(*

short summary
=============

.. <legal notes>

legal notes
=================
| SPDX-FileCopyrightText: © 2023 ekvip automation GmbH <info@ekvip.de>
| SPDX-License-Identifier: Apache-2.0
| For details check: Apache-2.0_

.. _Apache-2.0: https://www.apache.org/licenses/LICENSE-2.0

.. </legal notes>

methods and properties
======================

*)

{warning 'header is generated please add your documentation'}
FUNCTION_BLOCK StringAssertionTests EXTENDS AbstractAssertorTest

VAR
	testDataStringLengthIsExact 	: ARRAY[0 ..IsLengthTestDataSet.SIZE_OF_IS_DATASET] OF IsLengthBasicData;
	testDataStringContains 			: ARRAY[0..containsTestDataSet.SIZE_OF_CONTAINS_DATASET] OF containsDataStr;
	testDataStringContainsNo 		: ARRAY[0..containsNOTestDataSet.SIZE_OF_CONTAINSNO_DATASET] OF containsDataStr;
	testDataStringStartsWith		: ARRAY[0..startsWithDataSet.SIZE_OF_STARTWITH_DATASET] OF containsDataStr;
	testDataStringEndsWith 			: ARRAY[0..endsWithDataSet.SIZE_OF_ENDSWITH_DATASET] OF containsDataStr;
	testDataStringIsEqual			: ARRAY[0..isEqualToTestDataSet.SIZE_OF_ISEQUALTO_DATASET] OF isEqualToDataStr;
	testDataStringIsNotEqual		: ARRAY[0..isNotEqualToTestDataSet.SIZE_OF_ISNOTEQUALTO_DATASET] OF isEqualToDataStr;
	testDataStringIsEmpty			: ARRAY[0..isEmptyTestDataSet.SIZE_OF_ISEMPTY_DATASET] OF isEmptyDataStr;
	testDataStringIsNotEmpty		: ARRAY[0..isNotEmtyTestDataSet.SIZE_OF_ISNOTEMPTY_DATASET] OF isEmptyDataStr;
	testDataStringIsLenghtBetween	: ARRAY[0..IsLengthBetweenDataSet.SIZE_OF_LENGTHBETWEEN_DATASET] OF IsLengthBetweenBasicData;
	
END_VAR

testAnyString_isEmpty();
testAnyString_isNotEmpty();
testAnyString_isEqualTo();
testAnyString_isNotEqualTo();
testAnyString_lengthIsExact();


THIS^.runTestIsLength();
THIS^.runTestContains();
THIS^.runTestContainsNo();
THIS^.runTestEndsWith();
THIS^.runTestStartsWith();
THIS^.runTestIsEmpty();
THIS^.runTestIsNotEmpty();
THIS^.runTestIsEqualTo();
THIS^.runTestIsNotEqualTo();
THIS^.runTestLengthIsBetween();

(*

short summary
=============

.. <legal notes>

legal notes
=================
| SPDX-FileCopyrightText: © 2023 ekvip automation GmbH <info@ekvip.de>
| SPDX-License-Identifier: Apache-2.0
| For details check: Apache-2.0_

.. _Apache-2.0: https://www.apache.org/licenses/LICENSE-2.0

.. </legal notes>

parameters
==========

*)

{warning 'header is generated please add your documentation'}
METHOD FB_init : BOOL
VAR_INPUT
    bInitRetains : BOOL; // if TRUE, the retain variables are initialized (warm start / cold start)
    bInCopyCode : BOOL;  // if TRUE, the instance afterwards gets moved into the copy code (online change)
	classToBeTested :IAssertorContainer;
END_VAR
THIS^.testDataStringLengthIsExact 	:= IsLengthTestDataSet.IsLenghtDataSetCommon;
THIS^.testDataStringContains 		:= containsTestDataSet.containsDataSetCommon;	
THIS^.testDataStringContainsNo		:= containsNoTestDataSet.containsNoDataSetCommon;
THIS^.testDataStringEndsWith		:= endsWithDataSet.endsWithDataSetCommon;
THIS^.testDataStringStartsWith		:= startsWithDataSet.StartsWithDataSetCommon;
THIS^.testDataStringIsEqual			:= isEqualToTestDataSet.isEqualToDataSetCommon;		
THIS^.testDataStringIsNotEqual		:= isNotEqualToTestDataSet.isNotEqualDataSetCommon;
THIS^.testDataStringIsEmpty			:= isEmptyTestDataSet.isEmptyDataSetCommon;
THIS^.testDataStringIsNotEmpty		:= isNotEmtyTestDataSet.isNotEmptyDataSetCommon;
THIS^.testDataStringIsLenghtBetween	:= IsLengthBetweenDataSet.isLenghtBetweenToDataSetCommon;
END_METHOD

(*

short summary
=============

.. <legal notes>

legal notes
=================
| SPDX-FileCopyrightText: © 2023 ekvip automation GmbH <info@ekvip.de>
| SPDX-License-Identifier: Apache-2.0
| For details check: Apache-2.0_

.. _Apache-2.0: https://www.apache.org/licenses/LICENSE-2.0

.. </legal notes>

parameters
==========

*)

{warning 'header is generated please add your documentation'}
METHOD reset
VAR_INPUT
END_VAR
THIS^.assertorContainer.resetAssertor();
END_METHOD

(*

short summary
=============

.. <legal notes>

legal notes
=================
| SPDX-FileCopyrightText: © 2023 ekvip automation GmbH <info@ekvip.de>
| SPDX-License-Identifier: Apache-2.0
| For details check: Apache-2.0_

.. _Apache-2.0: https://www.apache.org/licenses/LICENSE-2.0

.. </legal notes>

parameters
==========

*)

{warning 'header is generated please add your documentation'}
METHOD runTestContains
VAR
	testDataIterator	:USINT;
END_VAR
TEST('ContainsTests');
FOR testDataIterator := 0 TO containsTestDataSet.SIZE_OF_contains_DATASET DO
	IF (THIS^.testDataStringContains[testDataIterator].typeToTest = TypeToTest.TEST_STRING) THEN
		
		THIS^.testAnyStringContains(THIS^.testDataStringContains[testDataIterator], testDataIterator);
		THIS^.testAsciiStringContains (THIS^.testDataStringContains[testDataIterator], testDataIterator);
		
	ELSIF (THIS^.testDataStringContains[testDataIterator].typeToTest = TypeToTest.TEST_WSTRING) THEN
		
		THIS^.testAnyStringContains(THIS^.testDataStringContains[testDataIterator], testDataIterator);
		THIS^.testUtf16StringContains(THIS^.testDataStringContains[testDataIterator], testDataIterator);
		
	END_IF;
END_FOR

TEST_FINISHED();
END_METHOD

(*

short summary
=============

.. <legal notes>

legal notes
=================
| SPDX-FileCopyrightText: © 2023 ekvip automation GmbH <info@ekvip.de>
| SPDX-License-Identifier: Apache-2.0
| For details check: Apache-2.0_

.. _Apache-2.0: https://www.apache.org/licenses/LICENSE-2.0

.. </legal notes>

parameters
==========

*)

{warning 'header is generated please add your documentation'}
METHOD runTestContainsNo
VAR
	testDataIterator	:USINT;
END_VAR
TEST('ContainsNoTests');
FOR testDataIterator:= 0 TO containsNoTestDataSet.SIZE_OF_containsNo_DATASET DO
	IF (THIS^.testDataStringContainsNo[testDataIterator].typeToTest = TypeToTest.TEST_STRING) THEN
		
		THIS^.testAnyStringContainsNo(THIS^.testDataStringContainsno[testDataIterator], testDataIterator);
		THIS^.testAsciiStringContainsNo (THIS^.testDataStringContainsno[testDataIterator], testDataIterator);
		
	ELSIF (THIS^.testDataStringContainsNo[testDataIterator].typeToTest = TypeToTest.TEST_WSTRING) THEN
		
		THIS^.testAnyStringContainsNo(THIS^.testDataStringContainsno[testDataIterator], testDataIterator);
		THIS^.testUtf16StringContainsNo(THIS^.testDataStringContainsno[testDataIterator], testDataIterator);
		
	END_IF;
END_FOR

TEST_FINISHED();
END_METHOD

(*

short summary
=============

.. <legal notes>

legal notes
=================
| SPDX-FileCopyrightText: © 2023 ekvip automation GmbH <info@ekvip.de>
| SPDX-License-Identifier: Apache-2.0
| For details check: Apache-2.0_

.. _Apache-2.0: https://www.apache.org/licenses/LICENSE-2.0

.. </legal notes>

parameters
==========

*)

{warning 'header is generated please add your documentation'}
METHOD runTestEndsWith
VAR
	testDataIterator	: USINT;
END_VAR
TEST('endsWithTests');

FOR testDataIterator := 0 TO endsWithDataSet.SIZE_OF_ENDSWITH_DATASET DO
	IF (THIS^.testDataStringEndsWith[testDataIterator].typeToTest = TypeToTest.TEST_STRING) THEN
		
		THIS^.testAnyStringEndsWith(THIS^.testDataStringEndsWith[testDataIterator], testDataIterator);
		THIS^.testAsciiEndsWith(THIS^.testDataStringEndsWith[testDataIterator], testDataIterator);
		
	ELSIF (THIS^.testDataStringEndsWith[testDataIterator].typeToTest = TypeToTest.TEST_WSTRING) THEN
		
		THIS^.testAnyStringEndsWith(THIS^.testDataStringEndsWith[testDataIterator], testDataIterator);
		THIS^.testUtf16EndsWith(THIS^.testDataStringEndsWith[testDataIterator], testDataIterator);
		
	END_IF;
END_FOR

TEST_FINISHED();
END_METHOD

(*

short summary
=============

.. <legal notes>

legal notes
=================
| SPDX-FileCopyrightText: © 2023 ekvip automation GmbH <info@ekvip.de>
| SPDX-License-Identifier: Apache-2.0
| For details check: Apache-2.0_

.. _Apache-2.0: https://www.apache.org/licenses/LICENSE-2.0

.. </legal notes>

parameters
==========

*)

{warning 'header is generated please add your documentation'}
METHOD runTestIsEmpty
VAR
	testDataIterator	: USINT;
END_VAR
TEST('isEmptyTests');

FOR testDataIterator := 0 TO isEmptyTestDataSet.SIZE_OF_ISEMPTY_DATASET DO
	IF (THIS^.testDataStringIsEmpty[testDataIterator].typeToTest = TypeToTest.TEST_STRING) THEN
		
		THIS^.testAnyStringIsEmpty(THIS^.testDataStringIsEmpty[testDataIterator], testDataIterator);
		THIS^.testAsciiIsEmpty(THIS^.testDataStringIsEmpty[testDataIterator], testDataIterator);
		
	ELSIF (THIS^.testDataStringIsEmpty[testDataIterator].typeToTest = TypeToTest.TEST_WSTRING) THEN
		
		THIS^.testAnyStringIsEmpty(THIS^.testDataStringIsEmpty[testDataIterator], testDataIterator);
		THIS^.testUtf16IsEmpty(THIS^.testDataStringIsEmpty[testDataIterator], testDataIterator);
		
	END_IF;
END_FOR

TEST_FINISHED();
END_METHOD

(*

short summary
=============

.. <legal notes>

legal notes
=================
| SPDX-FileCopyrightText: © 2023 ekvip automation GmbH <info@ekvip.de>
| SPDX-License-Identifier: Apache-2.0
| For details check: Apache-2.0_

.. _Apache-2.0: https://www.apache.org/licenses/LICENSE-2.0

.. </legal notes>

parameters
==========

*)

{warning 'header is generated please add your documentation'}
METHOD runTestIsEqualTo
VAR
	testDataIterator	: USINT;
END_VAR
TEST('isEqualToTests');

FOR testDataIterator := 0 TO isEqualToTestDataSet.SIZE_OF_ISEQUALTO_DATASET DO
	IF (THIS^.testDataStringIsEqual[testDataIterator].typeToTest = TypeToTest.TEST_STRING) THEN
		
		THIS^.testAnyStringIsEqualTo(THIS^.testDataStringIsEqual[testDataIterator], testDataIterator);
		THIS^.testAsciiIsEqualTo(THIS^.testDataStringIsEqual[testDataIterator], testDataIterator);
		
	ELSIF (THIS^.testDataStringIsEqual[testDataIterator].typeToTest = TypeToTest.TEST_WSTRING) THEN
		
		THIS^.testAnyStringIsEqualTo(THIS^.testDataStringIsEqual[testDataIterator], testDataIterator);
		THIS^.testUtf16IsEqualTo(THIS^.testDataStringIsEqual[testDataIterator], testDataIterator);
		
	END_IF;
END_FOR

TEST_FINISHED();
END_METHOD

(*

short summary
=============

.. <legal notes>

legal notes
=================
| SPDX-FileCopyrightText: © 2023 ekvip automation GmbH <info@ekvip.de>
| SPDX-License-Identifier: Apache-2.0
| For details check: Apache-2.0_

.. _Apache-2.0: https://www.apache.org/licenses/LICENSE-2.0

.. </legal notes>

parameters
==========

*)

{warning 'header is generated please add your documentation'}
METHOD runTestIsLength
VAR
	testDataIterator	:USINT;
END_VAR
TEST('IsLenghtIsTests');
FOR testDataIterator:= 0 TO IsLengthTestDataSet.SIZE_OF_IS_DATASET DO
	IF (THIS^.testDataStringLengthIsExact[testDataIterator].typeToTest = TypeToTest.TEST_STRING) THEN
		
		THIS^.testAnyStringLengthIs(THIS^.testDataStringLengthIsExact[testDataIterator], testDataIterator);
		THIS^.testAsciiStringlengthIs (THIS^.testDataStringLengthIsExact[testDataIterator], testDataIterator);
		
	ELSIF (THIS^.testDataStringLengthIsExact[testDataIterator].typeToTest = TypeToTest.TEST_WSTRING) THEN
		
		THIS^.testAnyStringLengthIs(THIS^.testDataStringLengthIsExact[testDataIterator], testDataIterator);
		THIS^.testUtf16StringlengthIs(THIS^.testDataStringLengthIsExact[testDataIterator], testDataIterator);
		
	END_IF;
END_FOR

TEST_FINISHED();
END_METHOD

(*

short summary
=============

.. <legal notes>

legal notes
=================
| SPDX-FileCopyrightText: © 2023 ekvip automation GmbH <info@ekvip.de>
| SPDX-License-Identifier: Apache-2.0
| For details check: Apache-2.0_

.. _Apache-2.0: https://www.apache.org/licenses/LICENSE-2.0

.. </legal notes>

parameters
==========

*)

{warning 'header is generated please add your documentation'}
METHOD runTestIsNotEmpty
VAR
	testDataIterator	: USINT;
END_VAR
TEST('isNotEmptyTests');

FOR testDataIterator := 0 TO isNotEmtyTestDataSet.SIZE_OF_ISNOTEMPTY_DATASET DO
	IF (THIS^.testDataStringIsNotEmpty[testDataIterator].typeToTest = TypeToTest.TEST_STRING) THEN
		
		THIS^.testAnyStringIsNotEmpty(THIS^.testDataStringIsNotEmpty[testDataIterator], testDataIterator);
		THIS^.testAsciiIsNotEmpty(THIS^.testDataStringIsNotEmpty[testDataIterator], testDataIterator);
		
	ELSIF (THIS^.testDataStringIsNotEmpty[testDataIterator].typeToTest = TypeToTest.TEST_WSTRING) THEN
		
		THIS^.testAnyStringIsNotEmpty(THIS^.testDataStringIsNotEmpty[testDataIterator], testDataIterator);
		THIS^.testUtf16IsNotEmpty(THIS^.testDataStringIsNotEmpty[testDataIterator], testDataIterator);
		
	END_IF;
END_FOR

TEST_FINISHED();
END_METHOD

(*

short summary
=============

.. <legal notes>

legal notes
=================
| SPDX-FileCopyrightText: © 2023 ekvip automation GmbH <info@ekvip.de>
| SPDX-License-Identifier: Apache-2.0
| For details check: Apache-2.0_

.. _Apache-2.0: https://www.apache.org/licenses/LICENSE-2.0

.. </legal notes>

parameters
==========

*)

{warning 'header is generated please add your documentation'}
METHOD runTestIsNotEqualTo
VAR
	testDataIterator	: USINT;
END_VAR
TEST('isNotEqualToTests');

FOR testDataIterator := 0 TO isNotEqualToTestDataSet.SIZE_OF_ISNOTEQUALTO_DATASET DO
	IF (THIS^.testDataStringIsNotEqual[testDataIterator].typeToTest = TypeToTest.TEST_STRING) THEN
		
		THIS^.testAnyStringIsNotEqualTo(THIS^.testDataStringIsNotEqual[testDataIterator], testDataIterator);
		THIS^.testAsciiIsNotEqualTo(THIS^.testDataStringIsNotEqual[testDataIterator], testDataIterator);
		
	ELSIF (THIS^.testDataStringIsNotEqual[testDataIterator].typeToTest = TypeToTest.TEST_WSTRING) THEN
		
		THIS^.testAnyStringIsNotEqualTo(THIS^.testDataStringIsNotEqual[testDataIterator], testDataIterator);
		THIS^.testUtf16IsNotEqualTo(THIS^.testDataStringIsNotEqual[testDataIterator], testDataIterator);
		
	END_IF;
END_FOR

TEST_FINISHED();
END_METHOD

(*

short summary
=============

.. <legal notes>

legal notes
=================
| SPDX-FileCopyrightText: © 2023 ekvip automation GmbH <info@ekvip.de>
| SPDX-License-Identifier: Apache-2.0
| For details check: Apache-2.0_

.. _Apache-2.0: https://www.apache.org/licenses/LICENSE-2.0

.. </legal notes>

parameters
==========

*)

{warning 'header is generated please add your documentation'}
METHOD runTestLengthIsBetween : BOOL
VAR
	testDataIterator	:USINT;
END_VAR
TEST('IsLenghtBetweenTests');
FOR testDataIterator:= 0 TO IsLengthBetweenDataSet.SIZE_OF_LENGTHBETWEEN_DATASET DO
	IF (THIS^.testDataStringIsLenghtBetween[testDataIterator].typeToTest = TypeToTest.TEST_STRING) THEN
		
		THIS^.testAnyStringLengthBetween(THIS^.testDataStringIsLenghtBetween[testDataIterator], testDataIterator);
		THIS^.testAsciiStringLengthBetween (THIS^.testDataStringIsLenghtBetween[testDataIterator], testDataIterator);
		
	ELSIF (THIS^.testDataStringIsLenghtBetween[testDataIterator].typeToTest = TypeToTest.TEST_WSTRING) THEN
		
		THIS^.testAnyStringLengthBetween(THIS^.testDataStringIsLenghtBetween[testDataIterator], testDataIterator);
		THIS^.testUtf16StringLengthBetween(THIS^.testDataStringIsLenghtBetween[testDataIterator], testDataIterator);
		
	END_IF;
END_FOR

TEST_FINISHED();
END_METHOD

(*

short summary
=============

.. <legal notes>

legal notes
=================
| SPDX-FileCopyrightText: © 2023 ekvip automation GmbH <info@ekvip.de>
| SPDX-License-Identifier: Apache-2.0
| For details check: Apache-2.0_

.. _Apache-2.0: https://www.apache.org/licenses/LICENSE-2.0

.. </legal notes>

parameters
==========

*)

{warning 'header is generated please add your documentation'}
METHOD runTestStartsWith
VAR
	testDataIterator	: USINT;
END_VAR
TEST('StartsWithTests');
FOR testDataIterator := 0 TO startsWithDataSet.SIZE_OF_STARTWITH_DATASET DO
	IF (THIS^.testDataStringStartsWith[testDataIterator].typeToTest = TypeToTest.TEST_STRING) THEN
		
		THIS^.testAnyStringStartsWith(THIS^.testDataStringStartsWith[testDataIterator], testDataIterator);
		THIS^.testAsciiStartsWith(THIS^.testDataStringStartsWith[testDataIterator], testDataIterator);
		
	ELSIF (THIS^.testDataStringStartsWith[testDataIterator].typeToTest = TypeToTest.TEST_WSTRING) THEN
		
		THIS^.testAnyStringStartsWith(THIS^.testDataStringStartsWith[testDataIterator], testDataIterator);
		THIS^.testUtf16StartsWith(THIS^.testDataStringStartsWith[testDataIterator], testDataIterator);
		
	END_IF;
END_FOR

TEST_FINISHED();
END_METHOD

(*

short summary
=============

.. <legal notes>

legal notes
=================
| SPDX-FileCopyrightText: © 2023 ekvip automation GmbH <info@ekvip.de>
| SPDX-License-Identifier: Apache-2.0
| For details check: Apache-2.0_

.. _Apache-2.0: https://www.apache.org/licenses/LICENSE-2.0

.. </legal notes>

parameters
==========

*)

{warning 'header is generated please add your documentation'}
METHOD testAnyString_isEmpty

VAR 
  testString1: STRING(50);
  testString2: STRING;
  number: INT;
END_VAR

// anyStringAssertionTests.isEmpty Tests

//-------------------------------------------------------------------------------------------------------
TEST('anyStringAssertionTest.isEmpty with stringToCheck:= emptyString');

testString1:= '';
THIS^.assertorContainer.resetAssertor();
THIS^.assertorContainer.assertor.assert.strings.anyString.isEmpty(
  stringToCheck := testString1,
  message := ''
);
THIS^.AssertFalse(
	Condition := THIS^.assertorContainer.wasAssertionWrong,
	Message := 'anyStringAssertionTests.isEmpty assertion shall be wrong, stringToCheck:= emptyString '
);
TEST_FINISHED();

//-------------------------------------------------------------------------------------------------------

TEST('anyStringAssertionTest.isEmpty with stringToCheck:= space');

testString1:= ' ';
THIS^.assertorContainer.resetAssertor();
THIS^.assertorContainer.assertor.assert.strings.anyString.isEmpty(
  stringToCheck := testString1,
  message := ''
);
THIS^.AssertTrue(
	Condition := THIS^.assertorContainer.wasAssertionWrong,
	Message := 'anyStringAssertionTests.isEmpty assertion shall be wrong, stringToCheck:= just space'
);
TEST_FINISHED();

//-------------------------------------------------------------------------------------------------------

TEST('anyStringAssertionTest.isEmpty with stringToCheck:= point');

testString1:= '.';
THIS^.assertorContainer.resetAssertor();
THIS^.assertorContainer.assertor.assert.strings.anyString.isEmpty(
  stringToCheck := testString1,
  message := ''
);
THIS^.AssertTrue(
	Condition := THIS^.assertorContainer.wasAssertionWrong,
	Message := 'anyStringAssertionTests.isEmpty assertion shall be wrong, stringToCheck:= point'
);
TEST_FINISHED();

//-------------------------------------------------------------------------------------------------------

TEST('anyStringAssertionTest.isEmpty with stringToCheck:= emptyStringVar');

testString1:= testString2;
THIS^.assertorContainer.resetAssertor();
THIS^.assertorContainer.assertor.assert.strings.anyString.isEmpty(
  stringToCheck := testString1,
  message := ''
);
THIS^.AssertFalse(
	Condition := THIS^.assertorContainer.wasAssertionWrong,
	Message := 'anyStringAssertionTests.isEmpty assertion shall be wrong, stringToCheck:= emptyStringVar'
);
TEST_FINISHED();

//-------------------------------------------------------------------------------------------------------

TEST('anyStringAssertionTest.isEmpty with stringToCheck:= wierdString');

testString1:= 'sadhasdhasduhuiashdui';
THIS^.assertorContainer.resetAssertor();
THIS^.assertorContainer.assertor.assert.strings.anyString.isEmpty(
  stringToCheck := testString1,
  message := ''
);
THIS^.AssertTrue(
	Condition := THIS^.assertorContainer.wasAssertionWrong,
	Message := 'anyStringAssertionTests.isEmpty assertion shall be wrong, stringToCheck:= emptyStringVar'
);
TEST_FINISHED();

//-------------------------------------------------------------------------------------------------------

TEST('anyStringAssertionTest.isEmpty with stringToCheck:=   +gdjsnd.8959889mfknfji');

testString1:= '   +gdjsnd.8959889mfknfji';
THIS^.assertorContainer.resetAssertor();
THIS^.assertorContainer.assertor.assert.strings.anyString.isEmpty(
  stringToCheck := testString1,
  message := ''
);
THIS^.AssertTrue(
	Condition := THIS^.assertorContainer.wasAssertionWrong,
	Message := 'anyStringAssertionTests.isEmpty assertion shall be wrong, stringToCheck:= emptyStringVar'
);
TEST_FINISHED();

//-------------------------------------------------------------------------------------------------------

TEST('anyStringAssertionTest.isEmpty with stringToCheck:=   converted int');

testString1:= INT_TO_STRING(number);
THIS^.assertorContainer.resetAssertor();
THIS^.assertorContainer.assertor.assert.strings.anyString.isEmpty(
  stringToCheck := testString1,
  message := ''
);
THIS^.AssertTrue(
	Condition := THIS^.assertorContainer.wasAssertionWrong,
	Message := 'anyStringAssertionTests.isEmpty assertion shall be wrong, stringToCheck:=  converted int'
);
TEST_FINISHED();
END_METHOD

(*

short summary
=============

.. <legal notes>

legal notes
=================
| SPDX-FileCopyrightText: © 2023 ekvip automation GmbH <info@ekvip.de>
| SPDX-License-Identifier: Apache-2.0
| For details check: Apache-2.0_

.. _Apache-2.0: https://www.apache.org/licenses/LICENSE-2.0

.. </legal notes>

parameters
==========

*)

{warning 'header is generated please add your documentation'}
METHOD testAnyString_isEqualTo

VAR 
  testString1: STRING(50);
  testString2: STRING(30);
  testString3: WSTRING(50);
  testString4: STRING(50);
  testString5: WSTRING(400);
  testString6: WSTRING(400);
  number: INT;
END_VAR

// anyStringAssertionTests.isEqualTo Tests

//-------------------------------------------------------------------------------------------------------
TEST('anyStringAssertionTest.isEqualTo with stringToCheck:= emptyString , expected:= emptyString , ignoreCases:= TRUE ,');

THIS^.assertorContainer.resetAssertor();
THIS^.assertorContainer.assertor.assert.strings.anyString.isEqualTo(
  stringToCheck:= testString1 , 
  expected:= testString2 ,
  ignoreCases:= TRUE ,
  message:='' );
  
THIS^.AssertFalse(
	Condition := THIS^.assertorContainer.wasAssertionWrong,
	Message := 'anyStringAssertionTests.isEqualTo , stringToCheck:= emptyString , expected:= emptyString , ignoreCases:= TRUE '
);
TEST_FINISHED();

//-------------------------------------------------------------------------------------------------------
TEST('anyStringAssertionTest.isEqualTo with stringToCheck:= emptyString assign , expected:= emptyString assign , ignoreCases:= TRUE ,');

testString1:= '';
testString2:= '';

THIS^.assertorContainer.resetAssertor();
THIS^.assertorContainer.assertor.assert.strings.anyString.isEqualTo(
  stringToCheck:= testString1 , 
  expected:= testString2 ,
  ignoreCases:= TRUE ,
  message:='' );
  
THIS^.AssertFalse(
	Condition := THIS^.assertorContainer.wasAssertionWrong,
	Message := 'anyStringAssertionTests.isEqualTo , stringToCheck:= emptyString assign, expected:= emptyString assign , ignoreCases:= TRUE '
);
TEST_FINISHED();

//-------------------------------------------------------------------------------------------------------
TEST('anyStringAssertionTest.isEqualTo with stringToCheck:= abcd56ä² , expected:= abcd56ä2 , ignoreCases:= TRUE ,');

testString1:= 'abcd56ä²';
testString2:= 'abcd56ä2';

THIS^.assertorContainer.resetAssertor();
THIS^.assertorContainer.assertor.assert.strings.anyString.isEqualTo(
  stringToCheck:= testString1 , 
  expected:= testString2 ,
  ignoreCases:= TRUE ,
  message:='' );
  
THIS^.AssertTrue(
	Condition := THIS^.assertorContainer.wasAssertionWrong,
	Message := 'anyStringAssertionTests.isEqualTo assertion shall be wrong, stringToCheck:= abcd56ä²  , expected:= abcd56ä2 , ignoreCases:= TRUE'
);
TEST_FINISHED();


//-------------------------------------------------------------------------------------------------------
TEST('anyStringAssertionTest.isEqualTo with stringToCheck:= abcd56ä²  , expected:= abcd56ä2 , ignoreCases:= False ,');

testString1:= 'abcd56ä²';
testString2:= 'abcd56ä2';

THIS^.assertorContainer.resetAssertor();
THIS^.assertorContainer.assertor.assert.strings.anyString.isEqualTo(
  stringToCheck:= testString1 , 
  expected:= testString2 ,
  ignoreCases:= FALSE ,
  message:='' );
  
THIS^.AssertTrue(
	Condition := THIS^.assertorContainer.wasAssertionWrong,
	Message := 'anyStringAssertionTests.isEqualTo assertion shall be wrong, stringToCheck:= abcd56ä²  , expected:= abcd56ä2 , ignoreCases:= false'
);
TEST_FINISHED();

//-------------------------------------------------------------------------------------------------------
TEST('anyStringAssertionTest.isEqualTo with stringToCheck:= abc d56ä2  , expected:= abc  d56ä2 , ignoreCases:= TRUE ,');

testString1:= 'abc d56ä2';
testString2:= 'abc  d56ä2';

THIS^.assertorContainer.resetAssertor();
THIS^.assertorContainer.assertor.assert.strings.anyString.isEqualTo(
  stringToCheck:= testString1 , 
  expected:= testString2 ,
  ignoreCases:= TRUE ,
  message:='' );
  
THIS^.AssertTrue(
	Condition := THIS^.assertorContainer.wasAssertionWrong,
	Message := 'anyStringAssertionTests.isEqualTo , stringToCheck:= abc d56ä2  , expected:= abc  d56ä2 , ignoreCases:= TRUE ,'
);
TEST_FINISHED();

//-------------------------------------------------------------------------------------------------------
TEST('anyStringAssertionTest.isEqualTo with stringToCheck:= abcd56ä2&§ (string) , expected:= abcd56ä2&§ (wstring), ignoreCases:= TRUE ,');

testString1:= 'abcd56ä2&§';
testString3:= "abcd56ä2&§";

THIS^.assertorContainer.resetAssertor();
THIS^.assertorContainer.assertor.assert.strings.anyString.isEqualTo(
  stringToCheck:= testString1 , 
  expected:= testString3 ,
  ignoreCases:= TRUE ,
  message:='' );
  
THIS^.AssertTrue(
	Condition := THIS^.assertorContainer.wasAssertionWrong,
	Message := 'anyStringAssertionTests.isEqualTo stringToCheck:= abcd56ä2&§ (string) , expected:= abcd56ä2&§ (wstring) , ignoreCases:= TRUE'
);
TEST_FINISHED();

//-------------------------------------------------------------------------------------------------------
TEST('anyStringAssertionTest.isEqualTo with stringToCheck:= abcd56ä2&§ (string) , expected:= abcd56ä2&§ (converted string)   , ignoreCases:= TRUE ,');

testString1:= 'abcd56ä2&§';
testString3:= "abcd56ä2&§";
testString4:= WSTRING_TO_STRING(testString3);

THIS^.assertorContainer.resetAssertor();
THIS^.assertorContainer.assertor.assert.strings.anyString.isEqualTo(
  stringToCheck:= testString1 , 
  expected:= testString4 ,
  ignoreCases:= TRUE ,
  message:='' );
  
THIS^.AssertFalse(
	Condition := THIS^.assertorContainer.wasAssertionWrong,
	Message := 'anyStringAssertionTests.isEqualTo stringToCheck:= abcd56ä2&§ (string) , expected:= expected:= abcd56ä2&§ (converted string) , ignoreCases:= TRUE'
);
TEST_FINISHED();


//-------------------------------------------------------------------------------------------------------
TEST('anyStringAssertionTest.isEqualTo with stringToCheck:= abcd56ä2&§ (string) , expected:= AbBd56ä2&§ , ignoreCases:= False ,');

testString1:= 'abcd56ä2&§';
testString2:='AbCd56ä2&§';

THIS^.assertorContainer.resetAssertor();
THIS^.assertorContainer.assertor.assert.strings.anyString.isEqualTo(
  stringToCheck:= testString1 , 
  expected:= testString2 ,
  ignoreCases:= TRUE ,
  message:='' );
  
THIS^.AssertFalse(
	Condition := THIS^.assertorContainer.wasAssertionWrong,
	Message := 'anyStringAssertionTests.isEqualTo with stringToCheck:= abcd56ä2&§  , expected:= AbBd56ä2&§ , ignoreCases:= False'
);
TEST_FINISHED();


//-------------------------------------------------------------------------------------------------------
TEST('anyStringAssertionTest.isEqualTo with stringToCheck:= äbcd56ä2&§ , expected:= äbcd56ä2&§ , ignoreCases:= False ,');

testString1:= 'abcd56ä2&§';
testString4:='äbcd56ä2&§';

THIS^.assertorContainer.resetAssertor();
THIS^.assertorContainer.assertor.assert.strings.anyString.isEqualTo(
  stringToCheck:= testString1 , 
  expected:= testString4 ,
  ignoreCases:= FALSE ,
  message:='' );
  
THIS^.AssertTrue(
	Condition := THIS^.assertorContainer.wasAssertionWrong,
	Message := 'anyStringAssertionTests.isEqualTo with stringToCheck:= abcd56ä2&§  , expected:= äbcd56ä2&§ , ignoreCases:= False'
);
TEST_FINISHED();

//-------------------------------------------------------------------------------------------------------
TEST('anyStringAssertionTest.isEqualTo with stringToCheck:= strange stuff arabic russian , expected:= strange stuff arabic russian , ignoreCases:= False ,');

testString5:= "иди сюда кусок дерьма ဒီကိုလာပါ ၊ تعال إلى هنا يا قطعة من الهراء";
testString6:="иди сюда кусок дерьма ဒီကိုလာပါ ၊ تعال إلى هنا يا قطعة من الهراء";

THIS^.assertorContainer.resetAssertor();
THIS^.assertorContainer.assertor.assert.strings.anyString.isEqualTo(
  stringToCheck:= testString5 , 
  expected:= testString6 ,
  ignoreCases:= FALSE ,
  message:='' );
  
THIS^.AssertFalse(
	Condition := THIS^.assertorContainer.wasAssertionWrong,
	Message := 'anyStringAssertionTests.isEqualTo with stringToCheck:= strange stuff arabic russian  , expected:= strange stuff arabic russian , ignoreCases:= False'
);
TEST_FINISHED();

//-------------------------------------------------------------------------------------------------------
TEST('anyStringAssertionTest.isEqualTo with stringToCheck:= strange stuff arabic russian 1 , expected:= strange stuff arabic russian 2, ignoreCases:= False ,');

testString5:= "иди сюд кусок дерьма ဒီကိုလာပါ ၊ تعال إلى هنا يا قطعة من الهراء";
testString6:="иди сюда кусок дерьма ဒီကိုလာပါ ၊ تعال إلى هنا يا قطعة من الهراء";

THIS^.assertorContainer.resetAssertor();
THIS^.assertorContainer.assertor.assert.strings.anyString.isEqualTo(
  stringToCheck:= testString5 , 
  expected:= testString6 ,
  ignoreCases:= FALSE ,
  message:='' );
  
THIS^.AssertTrue(
	Condition := THIS^.assertorContainer.wasAssertionWrong,
	Message := 'anyStringAssertionTests.isEqualTo with stringToCheck:= strange stuff arabic russian  , expected:= strange stuff arabic russian , ignoreCases:= False'
);
TEST_FINISHED();

//-------------------------------------------------------------------------------------------------------

TEST('anyStringAssertionTest.isEqualTo with stringToCheck:= strange stuff arabic russian capital , expected:= strange stuff arabic russian , ignoreCases:= true ,');

testString5:= "иди сюда Кусок дерьма ဒီကိုလာပါ ၊ تعال إلى هنا يا قطعة من الهراء";
testString6:="иди сюда кусок дерьма ဒီကိုလာပါ ၊ تعال إلى هنا يا قطعة من الهراء";

THIS^.assertorContainer.resetAssertor();
THIS^.assertorContainer.assertor.assert.strings.anyString.isEqualTo(
  stringToCheck:= testString5 , 
  expected:= testString6 ,
  ignoreCases:= TRUE ,
  message:='' );
  
THIS^.AssertFalse(
	Condition := THIS^.assertorContainer.wasAssertionWrong,
	Message := 'anyStringAssertionTests.isEqualTo with stringToCheck:= strange stuff arabic russian  , expected:= strange stuff arabic russian , ignoreCases:= true'
);
TEST_FINISHED();
END_METHOD

(*

short summary
=============

.. <legal notes>

legal notes
=================
| SPDX-FileCopyrightText: © 2023 ekvip automation GmbH <info@ekvip.de>
| SPDX-License-Identifier: Apache-2.0
| For details check: Apache-2.0_

.. _Apache-2.0: https://www.apache.org/licenses/LICENSE-2.0

.. </legal notes>

parameters
==========

*)

{warning 'header is generated please add your documentation'}
METHOD testAnyString_isNotEmpty

VAR
  testString1: STRING(50);
  testString2: STRING; 
END_VAR

// anyStringAssertionTests.isNotEmpty Tests

//-------------------------------------------------------------------------------------------------------
TEST('anyStringAssertionTest.isNotEmpty with stringToCheck:= emptyString');


testString1:= '';
THIS^.assertorContainer.resetAssertor();
THIS^.assertorContainer.assertor.assert.strings.anyString.isNOtEmpty(
  stringToCheck := testString1,
  message := ''
);
THIS^.AssertTrue(
	Condition := THIS^.assertorContainer.wasAssertionWrong,
	Message := 'anyStringAssertionTests.isNotEmpty assertion shall be wrong, stringToCheck:= emptyString '
);
TEST_FINISHED();

//-------------------------------------------------------------------------------------------------------

TEST('anyStringAssertionTest.isNotEmpty with stringToCheck:= space');

testString1:= ' ';
THIS^.assertorContainer.resetAssertor();
THIS^.assertorContainer.assertor.assert.strings.anyString.isNotEmpty(
  stringToCheck := testString1,
  message := ''
);
THIS^.AssertFalse(
	Condition := THIS^.assertorContainer.wasAssertionWrong,
	Message := 'anyStringAssertionTests.isNotEmpty assertion shall be wrong, stringToCheck:= just space'
);
TEST_FINISHED();

//-------------------------------------------------------------------------------------------------------

TEST('anyStringAssertionTest.isNotEmpty with stringToCheck:= point');

testString1:= '.';
THIS^.assertorContainer.resetAssertor();
THIS^.assertorContainer.assertor.assert.strings.anyString.isNotEmpty(
  stringToCheck := testString1,
  message := ''
);
THIS^.AssertFalse(
	Condition := THIS^.assertorContainer.wasAssertionWrong,
	Message := 'anyStringAssertionTests.isNotEmpty assertion shall be wrong, stringToCheck:= point'
);
TEST_FINISHED();

//-------------------------------------------------------------------------------------------------------

TEST('anyStringAssertionTest.isNotEmpty with stringToCheck:= emptyStringVar');

testString1:= testString2;
THIS^.assertorContainer.resetAssertor();
THIS^.assertorContainer.assertor.assert.strings.anyString.isNotEmpty(
  stringToCheck := testString1,
  message := ''
);
THIS^.AssertTrue(
	Condition := THIS^.assertorContainer.wasAssertionWrong,
	Message := 'anyStringAssertionTests.isNotEmpty assertion shall be wrong, stringToCheck:= emptyStringVar'
);
TEST_FINISHED();

//-------------------------------------------------------------------------------------------------------

TEST('anyStringAssertionTest.isNotEmpty with stringToCheck:= wierdString');

testString1:= 'sadhasdhasduhuiashdui';
THIS^.assertorContainer.resetAssertor();
THIS^.assertorContainer.assertor.assert.strings.anyString.isNotEmpty(
  stringToCheck := testString1,
  message := ''
);
THIS^.AssertFalse(
	Condition := THIS^.assertorContainer.wasAssertionWrong,
	Message := 'anyStringAssertionTests.isNotEmpty assertion shall be wrong, stringToCheck:= emptyStringVar'
);
TEST_FINISHED();

//-------------------------------------------------------------------------------------------------------

TEST('anyStringAssertionTest.isNotEmpty with stringToCheck:=   +gdjsnd.8959889mfknfji');

testString1:= '   +gdjsnd.8959889mfknfji';
THIS^.assertorContainer.resetAssertor();
THIS^.assertorContainer.assertor.assert.strings.anyString.isNotEmpty(
  stringToCheck := testString1,
  message := ''
);
THIS^.AssertFalse(
	Condition := THIS^.assertorContainer.wasAssertionWrong,
	Message := 'anyStringAssertionTests.isNotEmpty assertion shall be wrong, stringToCheck:= emptyStringVar'
);
TEST_FINISHED();
END_METHOD

(*

short summary
=============

.. <legal notes>

legal notes
=================
| SPDX-FileCopyrightText: © 2023 ekvip automation GmbH <info@ekvip.de>
| SPDX-License-Identifier: Apache-2.0
| For details check: Apache-2.0_

.. _Apache-2.0: https://www.apache.org/licenses/LICENSE-2.0

.. </legal notes>

parameters
==========

*)

{warning 'header is generated please add your documentation'}
METHOD testAnyString_isNotEqualTo 

VAR 
  testString1: STRING(50);
  testString2: STRING(30);
  testString3: WSTRING(50);
  testString4: STRING(50);
  testString5: WSTRING(400);
  testString6: WSTRING(400);
  number: INT;
END_VAR

// anyStringAssertionTests.isNotEqualTo Tests

//-------------------------------------------------------------------------------------------------------
TEST('anyStringAssertionTest.isNotEqualTo with stringToCheck:= emptyString , unexpected:= emptyString , ignoreCases:= TRUE ,');

THIS^.assertorContainer.resetAssertor();
THIS^.assertorContainer.assertor.assert.strings.anyString.isNotEqualTo(
  stringToCheck:= testString1 , 
  unexpected:= testString2 ,
  ignoreCases:= TRUE ,
  message:='' );
  
THIS^.AssertTrue(
	Condition := THIS^.assertorContainer.wasAssertionWrong,
	Message := 'anyStringAssertionTests.isNotEqualTo , stringToCheck:= emptyString , unexpected:= emptyString , ignoreCases:= TRUE'
);
TEST_FINISHED();


//-------------------------------------------------------------------------------------------------------
TEST('anyStringAssertionTest.isNotEqualTo with stringToCheck:= emptyString assign , unexpected:= emptyString assign , ignoreCases:= TRUE');

testString1:= '';
testString2:= '';

THIS^.assertorContainer.resetAssertor();
THIS^.assertorContainer.assertor.assert.strings.anyString.isNotEqualTo(
  stringToCheck:= testString1 , 
  unexpected:= testString2 ,
  ignoreCases:= TRUE ,
  message:='' );  
  
  
THIS^.AssertTrue(
	Condition := THIS^.assertorContainer.wasAssertionWrong,
	Message := 'anyStringAssertionTests.isNotEqualTo , stringToCheck:= emptyString assign, unexpected:= emptyString assign , ignoreCases:= TRUE');
TEST_FINISHED();

//-------------------------------------------------------------------------------------------------------

TEST('anyStringAssertionTest.isNotEqualTo with stringToCheck:= abcd56ä² , unexpected:= abcd56ä2 , ignoreCases:= TRUE ,');

testString1:= 'abcd56ä²';
testString2:= 'abcd56ä2';

THIS^.assertorContainer.resetAssertor();
THIS^.assertorContainer.assertor.assert.strings.anyString.isNotEqualTo(
  stringToCheck:= testString1 , 
  unexpected:= testString2 ,
  ignoreCases:= TRUE ,
  message:='' );
  
THIS^.AssertFalse(
	Condition := THIS^.assertorContainer.wasAssertionWrong,
	Message := 'anyStringAssertionTests.isNotEqualTo assertion shall be wrong, stringToCheck:= abcd56ä²  , unexpected:= abcd56ä2 , ignoreCases:= TRUE'
);
TEST_FINISHED();


//-------------------------------------------------------------------------------------------------------
TEST('anyStringAssertionTest.isEmpty with stringToCheck:= abcd56ä2  , unexpected:= abcd56ä2 , ignoreCases:= False ,');

testString1:= 'abcd56ä2';
testString2:= 'abcd56ä2';

THIS^.assertorContainer.resetAssertor();
THIS^.assertorContainer.assertor.assert.strings.anyString.isNotEqualTo(
  stringToCheck:= testString1 , 
  unexpected:= testString2 ,
  ignoreCases:= FALSE ,
  message:='' );
  
THIS^.AssertTrue(
	Condition := THIS^.assertorContainer.wasAssertionWrong,
	Message := 'anyStringAssertionTests.isNotEqualTo assertion shall be wrong, stringToCheck:= abcd56ä2  , unexpected:= abcd56ä2 , ignoreCases:= false'
);
TEST_FINISHED();


//-------------------------------------------------------------------------------------------------------
TEST('anyStringAssertionTest.isNotEqualTo with stringToCheck:= abc d56ä2  , unexpected:= abc  d56ä2 , ignoreCases:= TRUE ,');

testString1:= 'abc d56ä2';
testString2:= 'abc  d56ä2';

THIS^.assertorContainer.resetAssertor();
THIS^.assertorContainer.assertor.assert.strings.anyString.isnotEqualTo(
  stringToCheck:= testString1 , 
  unexpected:= testString2 ,
  ignoreCases:= TRUE ,
  message:='' );
  
THIS^.AssertFalse(
	Condition := THIS^.assertorContainer.wasAssertionWrong,
	Message := 'anyStringAssertionTests.isNotEqualTo , stringToCheck:= abc d56ä2  , unexpected:= abc  d56ä2 , ignoreCases:= TRUE ,'
);
TEST_FINISHED();

//-------------------------------------------------------------------------------------------------------
TEST('anyStringAssertionTest.isNotEqualTo with stringToCheck:= abcd56ä2&§ (string) , unexpected:= abcd56ä2&§ (wstring), ignoreCases:= TRUE ,');

testString1:= 'abcd56ä2&§';
testString3:= "abcd56ä2&§";

THIS^.assertorContainer.resetAssertor();
THIS^.assertorContainer.assertor.assert.strings.anyString.isNotEqualTo(
  stringToCheck:= testString1 , 
  unexpected:= testString3 ,
  ignoreCases:= TRUE ,
  message:='' );
  
THIS^.AssertFalse(
	Condition := THIS^.assertorContainer.wasAssertionWrong,
	Message := 'anyStringAssertionTests.isNotEqualTo stringToCheck:= abcd56ä2&§ (string) , unexpected:= abcd56ä2&§ (wstring) , ignoreCases:= TRUE'
);
TEST_FINISHED();

//-------------------------------------------------------------------------------------------------------
TEST('anyStringAssertionTest.isNotEqualTo with stringToCheck:= abcd56ä2&§ (string) , unexpected:= abcd56ä2&§ (converted string)   , ignoreCases:= TRUE ,');

testString1:= 'abcd56ä2&§';
testString3:= "abcd56ä2&§";
testString4:= WSTRING_TO_STRING(testString3);

THIS^.assertorContainer.resetAssertor();
THIS^.assertorContainer.assertor.assert.strings.anyString.isNotEqualTo(
  stringToCheck:= testString1 , 
  unexpected:= testString4 ,
  ignoreCases:= TRUE ,
  message:='' );
  
THIS^.AssertTrue(
	Condition := THIS^.assertorContainer.wasAssertionWrong,
	Message := 'anyStringAssertionTests.isNotEqualTo stringToCheck:= abcd56ä2&§ (string) , unexpected:= abcd56ä2&§ (converted string) , ignoreCases:= TRUE'
);
TEST_FINISHED();



//-------------------------------------------------------------------------------------------------------
TEST('anyStringAssertionTest.isNotEqualTo with stringToCheck:= abcd56ä2&§ (string) , unexpected:= AbBd56ä2&§ , ignoreCases:= False ,');

testString1:= 'abcd56ä2&§';
testString2:='AbCd56ä2&§';

THIS^.assertorContainer.resetAssertor();
THIS^.assertorContainer.assertor.assert.strings.anyString.isNotEqualTo(
  stringToCheck:= testString1 , 
  unexpected:= testString2 ,
  ignoreCases:= TRUE ,
  message:='' );
  
THIS^.AssertTrue(
	Condition := THIS^.assertorContainer.wasAssertionWrong,
	Message := 'anyStringAssertionTests.isNotEqualTo with stringToCheck:= abcd56ä2&§  , unexpected:= AbBd56ä2&§ , ignoreCases:= False'
);
TEST_FINISHED();


//-------------------------------------------------------------------------------------------------------
TEST('anyStringAssertionTest.isNotEqualTo with stringToCheck:= äbcd56ä2&§ , unexpected:= äbcd56ä2&§ , ignoreCases:= False ,');

testString1:= 'abcd56ä2&§';
testString4:='äbcd56ä2&§';

THIS^.assertorContainer.resetAssertor();
THIS^.assertorContainer.assertor.assert.strings.anyString.isNotEqualTo(
  stringToCheck:= testString1 , 
  unexpected:= testString4 ,
  ignoreCases:= FALSE ,
  message:='' );
  
THIS^.AssertFalse(
	Condition := THIS^.assertorContainer.wasAssertionWrong,
	Message := 'anyStringAssertionTests.isNotEqualTo with stringToCheck:= abcd56ä2&§  , unexpected:= äbcd56ä2&§ , ignoreCases:= False'
);
TEST_FINISHED();


//-------------------------------------------------------------------------------------------------------
TEST('anyStringAssertionTest.isNotEqualTo with stringToCheck:= strangestuff arabic russian , unexpected:= strangestuff arabic russian , ignoreCases:= False ,');

testString5:= "иди сюда кусок дерьма ဒီကိုလာပါ ၊ تعال إلى هنا يا قطعة من الهراء";
testString6:="иди сюда кусок дерьма ဒီကိုလာပါ ၊ تعال إلى هنا يا قطعة من الهراء";

THIS^.assertorContainer.resetAssertor();
THIS^.assertorContainer.assertor.assert.strings.anyString.isNotEqualTo(
  stringToCheck:= testString5 , 
  unexpected:= testString6 ,
  ignoreCases:= FALSE ,
  message:='' );
  
THIS^.AssertTrue(
	Condition := THIS^.assertorContainer.wasAssertionWrong,
	Message := 'anyStringAssertionTests.isNotEqualTo with stringToCheck:= abcd56ä2&§  , unexpected:= äbcd56ä2&§ , ignoreCases:= False'
);
TEST_FINISHED();

//-------------------------------------------------------------------------------------------------------
TEST('anyStringAssertionTest.isNotEqualTo with stringToCheck:= strangestuff arabic russian , unexpected:= strangestuff arabic russian cap, ignoreCases:= False ,');

testString5:= "иди сюда кусок дерьма ဒီကိုလာပါ ၊ تعال إلى هنا يا قطعة من الهراء";
testString6:="иди сюда Кусок дерьма ဒီကိုလာပါ ၊ تعال إلى هنا يا قطعة من الهراء";

THIS^.assertorContainer.resetAssertor();
THIS^.assertorContainer.assertor.assert.strings.anyString.isNotEqualTo(
  stringToCheck:= testString5 , 
  unexpected:= testString6 ,
  ignoreCases:= FALSE ,
  message:='' );
  
THIS^.AssertFalse(
	Condition := THIS^.assertorContainer.wasAssertionWrong,
	Message := 'anyStringAssertionTests.isNotEqualTo with stringToCheck:= abcd56ä2&§  , unexpected:= äbcd56ä2&§ , ignoreCases:= False'
);
TEST_FINISHED();
END_METHOD

(*

short summary
=============

.. <legal notes>

legal notes
=================
| SPDX-FileCopyrightText: © 2023 ekvip automation GmbH <info@ekvip.de>
| SPDX-License-Identifier: Apache-2.0
| For details check: Apache-2.0_

.. _Apache-2.0: https://www.apache.org/licenses/LICENSE-2.0

.. </legal notes>

parameters
==========

*)

{warning 'header is generated please add your documentation'}
METHOD testAnyString_lengthIsExact

VAR
  testString1:STRING(50);
  length: UDINT;
END_VAR
// anyStringAssertionTests.lengthIsExact Tests

//----------------------------------------------------------------------------------------------------------------------------------------
TEST('anyStringAssertionTest.lenghtIsExact with stringToCheck:= EmptyString(50) , expectedLength:= 0');

length := 0;

THIS^.assertorContainer.resetAssertor();
THIS^.assertorContainer.assertor.assert.strings.anyString.lenghtIsExact( 
	stringToCheck	:=	testString1, 
	expectedLength	:=	length,
	message			:=	''             
);

THIS^.AssertFalse(
	Condition	:=	THIS^.assertorContainer.wasAssertionWrong,
	Message		:=	'anyStringAssertionTests.lenghtIsExact with stringToCheck:= EmptyString(50) , expectedLength:= 0'
);

TEST_FINISHED();

//----------------------------------------------------------------------------------------------------------------------------------------

TEST('anyStringAssertionTest.lenghtIsExact with stringToCheck:= Hello World , expectedLength:= 11');

length:= 11;
testString1:= 'Hello World';

THIS^.assertorContainer.resetAssertor();
THIS^.assertorContainer.assertor.assert.strings.anyString.lenghtIsExact( stringToCheck    :=    testString1    , 
                                                       expectedLength   :=    length         ,
                                                       message          :=    ''             ) ;
THIS^.AssertFalse(
	Condition := THIS^.assertorContainer.wasAssertionWrong,
	Message   := 'anyStringAssertionTests.lenghtIsExact with stringToCheck:= Hello World , expectedLength:= 11');

TEST_FINISHED();

//----------------------------------------------------------------------------------------------------------------------------------------

TEST('anyStringAssertionTest.lenghtIsExact with stringToCheck:= Привет, мир , expectedLength:= 11');

length:= 11;
testString1:= 'Привет, мир';

THIS^.assertorContainer.resetAssertor();
THIS^.assertorContainer.assertor.assert.strings.anyString.lenghtIsExact( stringToCheck    :=    testString1    , 
                                                       expectedLength   :=    11             ,
                                                       message          :=    ''             ) ;
THIS^.AssertFalse(
	Condition := THIS^.assertorContainer.wasAssertionWrong,
	Message   := 'anyStringAssertionTests.lenghtIsExact with stringToCheck:= Привет, мир , expectedLength:= 11');

TEST_FINISHED();

//----------------------------------------------------------------------------------------------------------------------------------------

TEST('anyStringAssertionTest.lenghtIsExact with stringToCheck:= 6 spaces , expectedLength:= 6');

length:=6;
testString1:= '      ';

THIS^.assertorContainer.resetAssertor();
THIS^.assertorContainer.assertor.assert.strings.anyString.lenghtIsExact( stringToCheck    :=    testString1    , 
                                                       expectedLength   :=    length         ,
                                                       message          :=    ''             ) ;
THIS^.AssertFalse(
	Condition := THIS^.assertorContainer.wasAssertionWrong,
	Message   := 'anyStringAssertionTests.lenghtIsExact with stringToCheck:= 6 spaces , expectedLength:= 6');

TEST_FINISHED();

//----------------------------------------------------------------------------------------------------------------------------------------

TEST('anyStringAssertionTest.lenghtIsExact with stringToCheck:= Привет, мир Hello , expectedLength:= 17');

length:=17;
testString1:= 'Привет, мир Hello';

THIS^.assertorContainer.resetAssertor();
THIS^.assertorContainer.assertor.assert.strings.anyString.lenghtIsExact( stringToCheck    :=    testString1    , 
                                                       expectedLength   :=    length         ,
                                                       message          :=    ''             ) ;
THIS^.AssertFalse(
	Condition := THIS^.assertorContainer.wasAssertionWrong,
	Message   := 'anyStringAssertionTests.lenghtIsExact with stringToCheck:= Привет, мир Hello , expectedLength:= 17');

TEST_FINISHED();

//----------------------------------------------------------------------------------------------------------------------------------------

TEST('anyStringAssertionTest.lenghtIsExact with stringToCheck:= Привет, мир Hello , expectedLength:= 15');

length:=15;
testString1:= 'Привет, мир Hello';

THIS^.assertorContainer.resetAssertor();
THIS^.assertorContainer.assertor.assert.strings.anyString.lenghtIsExact( stringToCheck    :=    testString1    , 
                                                       expectedLength   :=    length         ,
                                                       message          :=    ''             ) ;
THIS^.AssertTrue(
	Condition := THIS^.assertorContainer.wasAssertionWrong,
	Message   := 'anyStringAssertionTests.lenghtIsExact with stringToCheck:= Привет, мир Hello , expectedLength:= 17');

TEST_FINISHED();
END_METHOD

(*

short summary
=============

.. <legal notes>

legal notes
=================
| SPDX-FileCopyrightText: © 2023 ekvip automation GmbH <info@ekvip.de>
| SPDX-License-Identifier: Apache-2.0
| For details check: Apache-2.0_

.. _Apache-2.0: https://www.apache.org/licenses/LICENSE-2.0

.. </legal notes>

parameters
==========

*)

{warning 'header is generated please add your documentation'}
METHOD testAnyStringContains : BOOL
VAR_INPUT
	inputStruct	: containsDataStr;
	testNumber :USINT;

END_VAR

VAR
	message : STRING;
END_VAR
THIS^.reset();
	

IF (inputStruct.typeToTest = TypeToTest.TEST_WSTRING) THEN
	THIS^.assertorContainer.assertor.assert.strings.anyString.contains(
		stringToCheck 	:= inputStruct.WStringToTest,
		searchString	:= inputStruct.WStringToContain, 
		ignoreCases		:= inputStruct.IgnoreCases,
		message			:= ''
	);			
ELSIF  (inputStruct.typeToTest = TypeToTest.TEST_STRING ) THEN
	THIS^.assertorContainer.assertor.assert.strings.anyString.contains(
		stringToCheck 	:= inputStruct.StringToTest,
		searchString	:= inputStruct.StringToContain, 
		ignoreCases		:= inputStruct.IgnoreCases,
		message			:= ''
	);

END_IF

message	:= CONCAT( 'Test Number ', TO_STRING(testNumber));
message	:= CONCAT( message, ' during function AnyString.contains ');
message	:= CONCAT( Message , ' has failed ');

THIS^.AssertEquals_BOOL(
	Expected 	:= inputStruct.expectedResult,
	Actual 		:= THIS^.assertorContainer.wasAssertionWrong,
	Message 	:= message
);
END_METHOD

(*

short summary
=============

.. <legal notes>

legal notes
=================
| SPDX-FileCopyrightText: © 2023 ekvip automation GmbH <info@ekvip.de>
| SPDX-License-Identifier: Apache-2.0
| For details check: Apache-2.0_

.. _Apache-2.0: https://www.apache.org/licenses/LICENSE-2.0

.. </legal notes>

parameters
==========

*)

{warning 'header is generated please add your documentation'}
METHOD testAnyStringContainsNo : BOOL
VAR_INPUT
	inputStruct	: containsDataStr;
	testNumber 	: USINT;
END_VAR

VAR
	message : STRING;
END_VAR
THIS^.reset();

IF (inputStruct.typeToTest = TypeToTest.TEST_WSTRING) THEN
	THIS^.assertorContainer.assertor.assert.strings.anyString.containsNo(
		stringToCheck 	:= inputStruct.WStringToTest,
		searchString	:= inputStruct.WStringToContain, 
		ignoreCases		:= inputStruct.IgnoreCases,
		message			:= ''
	);
					
ELSIF  (inputStruct.typeToTest = TypeToTest.TEST_STRING ) THEN
	THIS^.assertorContainer.assertor.assert.strings.anyString.containsNo(
		stringToCheck 	:= inputStruct.StringToTest,
		searchString	:= inputStruct.StringToContain, 
		ignoreCases		:= inputStruct.IgnoreCases,
		message			:= ''
	);

END_IF

message	:= CONCAT( 'Test Number ', TO_STRING(testNumber));
message	:= CONCAT( message, ' during function AnyString.containsNo ');
message	:= CONCAT( Message , ' has failed ');

THIS^.AssertEquals_BOOL(
	Expected 	:= inputStruct.expectedResult,
	Actual 		:= THIS^.assertorContainer.wasAssertionWrong,
	Message 	:= message
);
END_METHOD

(*

short summary
=============

.. <legal notes>

legal notes
=================
| SPDX-FileCopyrightText: © 2023 ekvip automation GmbH <info@ekvip.de>
| SPDX-License-Identifier: Apache-2.0
| For details check: Apache-2.0_

.. _Apache-2.0: https://www.apache.org/licenses/LICENSE-2.0

.. </legal notes>

parameters
==========

*)

{warning 'header is generated please add your documentation'}
METHOD testAnyStringEndsWith : BOOL
VAR_INPUT
	inputStruct	: containsDataStr;
	testNumber 	: USINT;
END_VAR

VAR
	message : STRING;
END_VAR
THIS^.reset();

IF (inputStruct.typeToTest = TypeToTest.TEST_WSTRING) THEN
	THIS^.assertorContainer.assertor.assert.strings.anyString.endsWith(
		stringToCheck	:= inputStruct.WStringToTest,
		end				:= inputStruct.WStringToContain,
		ignoreCases		:= inputStruct.IgnoreCases,
		trim			:= inputStruct.Trim,
		message			:= ''
	);
					
ELSIF  (inputStruct.typeToTest = TypeToTest.TEST_STRING ) THEN
	THIS^.assertorContainer.assertor.assert.strings.anyString.endsWith(
		stringToCheck	:= inputStruct.StringToTest,
		end				:= inputStruct.StringToContain,
		ignoreCases		:= inputStruct.IgnoreCases,
		trim			:= inputStruct.Trim,
		message			:= ''
	);
	
END_IF

message	:= CONCAT( 'Test Number ', TO_STRING(testNumber));
message	:= CONCAT( message, ' during function AnyString.endsWith ');
message	:= CONCAT( Message , ' has failed ');

THIS^.AssertEquals_BOOL(
	Expected 	:= inputStruct.expectedResult,
	Actual 		:= THIS^.assertorContainer.wasAssertionWrong,
	Message 	:= message
);
END_METHOD

(*

short summary
=============

.. <legal notes>

legal notes
=================
| SPDX-FileCopyrightText: © 2023 ekvip automation GmbH <info@ekvip.de>
| SPDX-License-Identifier: Apache-2.0
| For details check: Apache-2.0_

.. _Apache-2.0: https://www.apache.org/licenses/LICENSE-2.0

.. </legal notes>

parameters
==========

*)

{warning 'header is generated please add your documentation'}
METHOD testAnyStringIsEmpty : BOOL
VAR_INPUT
	inputStruct	: isEmptyDataStr;
	testNumber 	: USINT;
END_VAR

VAR
	message : STRING;
END_VAR
THIS^.reset();

IF (inputStruct.typeToTest = TypeToTest.TEST_WSTRING) THEN
	THIS^.assertorContainer.assertor.assert.strings.anyString.isEmpty(
		stringToCheck 	:= inputStruct.WStringToTest,
		message			:= ''
	);
					
ELSIF  (inputStruct.typeToTest = TypeToTest.TEST_STRING ) THEN
	THIS^.assertorContainer.assertor.assert.strings.anyString.isEmpty(
		stringToCheck 	:= inputStruct.StringToTest,
		message			:= ''
	);
	
END_IF

message	:= CONCAT( 'Test Number ', TO_STRING(testNumber));
message	:= CONCAT( message, ' during function AnyString.isEmpty ');
message	:= CONCAT( Message , ' has failed ');

THIS^.AssertEquals_BOOL(
	Expected 	:= inputStruct.expectedResult,
	Actual 		:= THIS^.assertorContainer.wasAssertionWrong,
	Message 	:= message
);
END_METHOD

(*

short summary
=============

.. <legal notes>

legal notes
=================
| SPDX-FileCopyrightText: © 2023 ekvip automation GmbH <info@ekvip.de>
| SPDX-License-Identifier: Apache-2.0
| For details check: Apache-2.0_

.. _Apache-2.0: https://www.apache.org/licenses/LICENSE-2.0

.. </legal notes>

parameters
==========

*)

{warning 'header is generated please add your documentation'}
METHOD testAnyStringIsEqualTo : BOOL
VAR_INPUT
	inputStruct	: isEqualToDataStr;
	testNumber 	: USINT;
END_VAR

VAR
	message : STRING;
END_VAR
THIS^.reset();

IF (inputStruct.typeToTest = TypeToTest.TEST_WSTRING) THEN
	THIS^.assertorContainer.assertor.assert.strings.anyString.isEqualTo(
		stringToCheck 	:= inputStruct.WStringToTest,
		expected		:= inputStruct.EqualToWString,
		ignoreCases     := inputStruct.IgnoreCases,
		message			:= ''	 	
	);
					
ELSIF  (inputStruct.typeToTest = TypeToTest.TEST_STRING ) THEN
	THIS^.assertorContainer.assertor.assert.strings.anyString.isEqualTo(
		stringToCheck 	:= inputStruct.StringToTest,
		expected		:= inputStruct.EqualToString,
		ignoreCases     := inputStruct.IgnoreCases,
		message			:= ''
	);
	
END_IF

message	:= CONCAT( 'Test Number ', TO_STRING(testNumber));
message	:= CONCAT( message, ' during function AnyString.isEqualTo ');
message	:= CONCAT( Message , ' has failed ');

THIS^.AssertEquals_BOOL(
	Expected 	:= inputStruct.expectedResult,
	Actual 		:= THIS^.assertorContainer.wasAssertionWrong,
	Message 	:= message
);
END_METHOD

(*

short summary
=============

.. <legal notes>

legal notes
=================
| SPDX-FileCopyrightText: © 2023 ekvip automation GmbH <info@ekvip.de>
| SPDX-License-Identifier: Apache-2.0
| For details check: Apache-2.0_

.. _Apache-2.0: https://www.apache.org/licenses/LICENSE-2.0

.. </legal notes>

parameters
==========

*)

{warning 'header is generated please add your documentation'}
METHOD testAnyStringIsNotEmpty : BOOL
VAR_INPUT
	inputStruct	: isEmptyDataStr;
	testNumber 	: USINT;
END_VAR

VAR
	message : STRING;
END_VAR
THIS^.reset();

IF (inputStruct.typeToTest = TypeToTest.TEST_WSTRING) THEN
	THIS^.assertorContainer.assertor.assert.strings.anyString.isNotEmpty(
		stringToCheck 	:= inputStruct.WStringToTest,
		message			:= ''
	);
					
ELSIF  (inputStruct.typeToTest = TypeToTest.TEST_STRING ) THEN
	THIS^.assertorContainer.assertor.assert.strings.anyString.isNotEmpty(
		stringToCheck 	:= inputStruct.StringToTest,
		message			:= ''
	);
	
END_IF

message	:= CONCAT( 'Test Number ', TO_STRING(testNumber));
message	:= CONCAT( message, ' during function AnyString.isNotEmpty ');
message	:= CONCAT( Message , ' has failed ');

THIS^.AssertEquals_BOOL(
	Expected 	:= inputStruct.expectedResult,
	Actual 		:= THIS^.assertorContainer.wasAssertionWrong,
	Message 	:= message
);
END_METHOD

(*

short summary
=============

.. <legal notes>

legal notes
=================
| SPDX-FileCopyrightText: © 2023 ekvip automation GmbH <info@ekvip.de>
| SPDX-License-Identifier: Apache-2.0
| For details check: Apache-2.0_

.. _Apache-2.0: https://www.apache.org/licenses/LICENSE-2.0

.. </legal notes>

parameters
==========

*)

{warning 'header is generated please add your documentation'}
METHOD testAnyStringIsNotEqualTo : BOOL
VAR_INPUT
	inputStruct	: isEqualToDataStr;
	testNumber 	: USINT;
END_VAR

VAR
	message : STRING;
END_VAR
THIS^.reset();

IF (inputStruct.typeToTest = TypeToTest.TEST_WSTRING) THEN
	THIS^.assertorContainer.assertor.assert.strings.anyString.isNotEqualTo(
		stringToCheck 	:= inputStruct.WStringToTest,
		unexpected		:= inputStruct.EqualToWString,
		ignoreCases     := inputStruct.IgnoreCases,
		message			:= ''	 	
	);
					
ELSIF  (inputStruct.typeToTest = TypeToTest.TEST_STRING ) THEN
	THIS^.assertorContainer.assertor.assert.strings.anyString.isNotEqualTo(
		stringToCheck 	:= inputStruct.StringToTest,
		unexpected		:= inputStruct.EqualToString,
		ignoreCases     := inputStruct.IgnoreCases,
		message			:= ''
	);
	
END_IF

message	:= CONCAT( 'Test Number ', TO_STRING(testNumber));
message	:= CONCAT( message, ' during function AnyString.isNotEqualTo ');
message	:= CONCAT( Message , ' has failed ');

THIS^.AssertEquals_BOOL(
	Expected 	:= inputStruct.expectedResult,
	Actual 		:= THIS^.assertorContainer.wasAssertionWrong,
	Message 	:= message
);
END_METHOD

(*

short summary
=============

.. <legal notes>

legal notes
=================
| SPDX-FileCopyrightText: © 2023 ekvip automation GmbH <info@ekvip.de>
| SPDX-License-Identifier: Apache-2.0
| For details check: Apache-2.0_

.. _Apache-2.0: https://www.apache.org/licenses/LICENSE-2.0

.. </legal notes>

parameters
==========

*)

{warning 'header is generated please add your documentation'}
METHOD testAnyStringLengthBetween
VAR_INPUT
	inputStruct	: IsLengthBetweenBasicData;
	testNumber	: USINT;
END_VAR

VAR
	message	: STRING;
END_VAR

THIS^.reset();

IF (inputStruct.typeToTest = TypeToTest.TEST_WSTRING) THEN	
	THIS^.assertorContainer.assertor.assert.strings.anyString.lenghtIsBetween( 
		stringToCheck	:=	inputStruct.wstringToTest, 
		maxLenght		:=	inputStruct.maxLength,
		minLenght   	:=  inputStruct.minLength,
		message			:=	''          
	);
				
ELSIF  (inputStruct.typeToTest = TypeToTest.TEST_STRING ) THEN
    THIS^.assertorContainer.assertor.assert.strings.anyString.lenghtIsBetween( 
		stringToCheck	:=	inputStruct.stringToTest, 
		maxLenght		:=	inputStruct.maxLength,
		minLenght   	:=  inputStruct.minLength,
		message			:=	''          
	);
END_IF

message	:= CONCAT( 'Test Number ', TO_STRING(testNumber));
message	:= CONCAT( message, ' during function AnyString.isLengthBetween ');
message	:= CONCAT( Message , ' has failed ');
	
THIS^.AssertEquals_BOOL(
	Expected 	:= inputStruct.expectedResult,
	Actual 		:= THIS^.assertorContainer.wasAssertionWrong,
	Message 	:= message
);
	
//TEST_FINISHED();
END_METHOD

(*

short summary
=============

.. <legal notes>

legal notes
=================
| SPDX-FileCopyrightText: © 2023 ekvip automation GmbH <info@ekvip.de>
| SPDX-License-Identifier: Apache-2.0
| For details check: Apache-2.0_

.. _Apache-2.0: https://www.apache.org/licenses/LICENSE-2.0

.. </legal notes>

parameters
==========

*)

{warning 'header is generated please add your documentation'}
METHOD testAnyStringLengthIs
VAR_INPUT
	inputStruct	:IsLengthBasicData;
	testNumber :USINT;
END_VAR

VAR
	message: STRING;
END_VAR


THIS^.reset();

IF (inputStruct.typeToTest = TypeToTest.TEST_WSTRING) THEN
	IF (inputStruct.funcType = FunctionType.EXACT) THEN 
		THIS^.assertorContainer.assertor.assert.strings.anyString.lenghtIsExact( 
			stringToCheck	:=	inputStruct.wstringToTest, 
			expectedLength	:=	inputStruct.expectedLength,
			message			:=	''          
		);
	ELSIF (inputStruct.funcType = FunctionType.MAXIMUM) THEN
		THIS^.assertorContainer.assertor.assert.strings.anyString.lenghtIsMax( 
			stringToCheck	:=	inputStruct.wstringToTest, 
			maxLength		:=	inputStruct.expectedLength,
			message			:=	''
		);
	ELSIF (inputStruct.funcType = FunctionType.MINIMUM) THEN
		THIS^.assertorContainer.assertor.assert.strings.anyString.lenghtIsMin( 
			stringToCheck	:=	inputStruct.wstringToTest, 
			minLength		:=	inputStruct.expectedLength,
			message			:=	''
		);
	END_IF;
				
ELSIF  (inputStruct.typeToTest = TypeToTest.TEST_STRING ) THEN
    IF (inputStruct.funcType = FunctionType.EXACT) THEN 
		THIS^.assertorContainer.assertor.assert.strings.anyString.lenghtIsExact( 
			stringToCheck	:=	inputStruct.stringToTest, 
			expectedLength	:=	inputStruct.expectedLength,
			message			:=	''         
		);
	ELSIF (inputStruct.funcType = FunctionType.MAXIMUM) THEN
		THIS^.assertorContainer.assertor.assert.strings.anyString.lenghtIsMax( 
			stringToCheck	:=	inputStruct.stringToTest, 
			maxLength		:=	inputStruct.expectedLength,
			message			:=	''        
		);
	ELSIF (inputStruct.funcType = FunctionType.MINIMUM) THEN
		THIS^.assertorContainer.assertor.assert.strings.anyString.lenghtIsMin( 
			stringToCheck	:=	inputStruct.stringToTest, 
			minLength		:=	inputStruct.expectedLength,
			message			:=	''          
		);
	END_IF;

END_IF

message	:= CONCAT( 'Test Number ', TO_STRING(testNumber));
message	:= CONCAT( message, ' during function AnyString.isLength ');
message	:= CONCAT( message , TO_STRING(inputStruct.funcType));
message	:= CONCAT( Message , ' has failed ');
	
THIS^.AssertEquals_BOOL(
	Expected 	:= inputStruct.expectedResult,
	Actual 		:= THIS^.assertorContainer.wasAssertionWrong,
	Message 	:= message
);
	
//TEST_FINISHED();
END_METHOD

(*

short summary
=============

.. <legal notes>

legal notes
=================
| SPDX-FileCopyrightText: © 2023 ekvip automation GmbH <info@ekvip.de>
| SPDX-License-Identifier: Apache-2.0
| For details check: Apache-2.0_

.. _Apache-2.0: https://www.apache.org/licenses/LICENSE-2.0

.. </legal notes>

parameters
==========

*)

{warning 'header is generated please add your documentation'}
METHOD testAnyStringStartsWith : BOOL
VAR_INPUT
	inputStruct	: containsDataStr;
	testNumber 	: USINT;
END_VAR

VAR
	message : STRING;
END_VAR
THIS^.reset();

IF (inputStruct.typeToTest = TypeToTest.TEST_WSTRING) THEN
	THIS^.assertorContainer.assertor.assert.strings.anyString.startsWith(
		stringToCheck	:= inputStruct.WStringToTest,
		start			:= inputStruct.WStringToContain,
		ignoreCases		:= inputStruct.IgnoreCases,
		trim			:= inputStruct.Trim,
		message			:= ''
	);
					
ELSIF  (inputStruct.typeToTest = TypeToTest.TEST_STRING ) THEN
	THIS^.assertorContainer.assertor.assert.strings.anyString.startsWith(
		stringToCheck	:= inputStruct.StringToTest,
		start			:= inputStruct.StringToContain,
		ignoreCases		:= inputStruct.IgnoreCases,
		trim			:= inputStruct.Trim,
		message			:= ''
	);

END_IF

message	:= CONCAT( 'Test Number ', TO_STRING(testNumber));
message	:= CONCAT( message, ' during function AnyString.startsWith ');
message	:= CONCAT( Message , ' has failed ');

THIS^.AssertEquals_BOOL(
	Expected 	:= inputStruct.expectedResult,
	Actual 		:= THIS^.assertorContainer.wasAssertionWrong,
	Message 	:= message
);
END_METHOD

(*

short summary
=============

.. <legal notes>

legal notes
=================
| SPDX-FileCopyrightText: © 2023 ekvip automation GmbH <info@ekvip.de>
| SPDX-License-Identifier: Apache-2.0
| For details check: Apache-2.0_

.. _Apache-2.0: https://www.apache.org/licenses/LICENSE-2.0

.. </legal notes>

parameters
==========

*)

{warning 'header is generated please add your documentation'}
METHOD testAsciiEndsWith : BOOL
VAR_INPUT
	inputStruct	: containsDataStr;
	testNumber 	: USINT;
END_VAR

VAR
	message : STRING;
END_VAR
THIS^.reset();

THIS^.assertorContainer.assertor.assert.strings.ascii.endsWith(
	stringToCheck	:= inputStruct.StringToTest,
	end				:= inputStruct.StringToContain,
	ignoreCases		:= inputStruct.IgnoreCases,
	trim			:= inputStruct.Trim,
	message			:= ''
);


message	:= CONCAT( 'Test Number ', TO_STRING(testNumber));
message	:= CONCAT( message, ' during function Ascii.endsWith ');
message	:= CONCAT( Message , ' has failed ');

THIS^.AssertEquals_BOOL(
	Expected 	:= inputStruct.expectedResult,
	Actual 		:= THIS^.assertorContainer.wasAssertionWrong,
	Message 	:= message
);
END_METHOD

(*

short summary
=============

.. <legal notes>

legal notes
=================
| SPDX-FileCopyrightText: © 2023 ekvip automation GmbH <info@ekvip.de>
| SPDX-License-Identifier: Apache-2.0
| For details check: Apache-2.0_

.. _Apache-2.0: https://www.apache.org/licenses/LICENSE-2.0

.. </legal notes>

parameters
==========

*)

{warning 'header is generated please add your documentation'}
METHOD testAsciiIsEmpty : BOOL
VAR_INPUT
	inputStruct	: isEmptyDataStr;
	testNumber 	: USINT;
END_VAR

VAR
	message : STRING;
END_VAR
THIS^.reset();

THIS^.assertorContainer.assertor.assert.strings.anyString.isEmpty(
	stringToCheck 	:= inputStruct.StringToTest,
	message			:= ''
);

message	:= CONCAT( 'Test Number ', TO_STRING(testNumber));
message	:= CONCAT( message, ' during function Ascii.isEmpty ');
message	:= CONCAT( Message , ' has failed ');

THIS^.AssertEquals_BOOL(
	Expected 	:= inputStruct.expectedResult,
	Actual 		:= THIS^.assertorContainer.wasAssertionWrong,
	Message 	:= message
);
END_METHOD

(*

short summary
=============

.. <legal notes>

legal notes
=================
| SPDX-FileCopyrightText: © 2023 ekvip automation GmbH <info@ekvip.de>
| SPDX-License-Identifier: Apache-2.0
| For details check: Apache-2.0_

.. _Apache-2.0: https://www.apache.org/licenses/LICENSE-2.0

.. </legal notes>

parameters
==========

*)

{warning 'header is generated please add your documentation'}
METHOD testAsciiIsEqualTo : BOOL
VAR_INPUT
	inputStruct	: isEqualToDataStr;
	testNumber 	: USINT;
END_VAR

VAR
	message : STRING;
END_VAR
THIS^.reset();

THIS^.assertorContainer.assertor.assert.strings.ascii.isEqualTo(
	stringToCheck 	:= inputStruct.StringToTest,
	expected		:= inputStruct.EqualToString,
	ignoreCases     := inputStruct.IgnoreCases,
	message			:= ''	 	
);

message	:= CONCAT( 'Test Number ', TO_STRING(testNumber));
message	:= CONCAT( message, ' during function Ascii.isEqualTo ');
message	:= CONCAT( Message , ' has failed ');

THIS^.AssertEquals_BOOL(
	Expected 	:= inputStruct.expectedResult,
	Actual 		:= THIS^.assertorContainer.wasAssertionWrong,
	Message 	:= message
);
END_METHOD

(*

short summary
=============

.. <legal notes>

legal notes
=================
| SPDX-FileCopyrightText: © 2023 ekvip automation GmbH <info@ekvip.de>
| SPDX-License-Identifier: Apache-2.0
| For details check: Apache-2.0_

.. _Apache-2.0: https://www.apache.org/licenses/LICENSE-2.0

.. </legal notes>

parameters
==========

*)

{warning 'header is generated please add your documentation'}
METHOD testAsciiIsNotEmpty : BOOL
VAR_INPUT
	inputStruct	: isEmptyDataStr;
	testNumber 	: USINT;
END_VAR

VAR
	message : STRING;
END_VAR
THIS^.reset();

THIS^.assertorContainer.assertor.assert.strings.anyString.isNotEmpty(
	stringToCheck 	:= inputStruct.StringToTest,
	message			:= ''
);

message	:= CONCAT( 'Test Number ', TO_STRING(testNumber));
message	:= CONCAT( message, ' during function Ascii.isNotEmpty ');
message	:= CONCAT( Message , ' has failed ');

THIS^.AssertEquals_BOOL(
	Expected 	:= inputStruct.expectedResult,
	Actual 		:= THIS^.assertorContainer.wasAssertionWrong,
	Message 	:= message
);
END_METHOD

(*

short summary
=============

.. <legal notes>

legal notes
=================
| SPDX-FileCopyrightText: © 2023 ekvip automation GmbH <info@ekvip.de>
| SPDX-License-Identifier: Apache-2.0
| For details check: Apache-2.0_

.. _Apache-2.0: https://www.apache.org/licenses/LICENSE-2.0

.. </legal notes>

parameters
==========

*)

{warning 'header is generated please add your documentation'}
METHOD testAsciiIsNotEqualTo : BOOL
VAR_INPUT
	inputStruct	: isEqualToDataStr;
	testNumber 	: USINT;
END_VAR

VAR
	message : STRING;
END_VAR
THIS^.reset();

THIS^.assertorContainer.assertor.assert.strings.anyString.isNotEqualTo(
	stringToCheck 	:= inputStruct.StringToTest,
	unexpected		:= inputStruct.EqualToString,
	ignoreCases     := inputStruct.IgnoreCases,
	message			:= ''	 	
);

message	:= CONCAT( 'Test Number ', TO_STRING(testNumber));
message	:= CONCAT( message, ' during function Ascii.isNotEqualTo ');
message	:= CONCAT( Message , ' has failed ');

THIS^.AssertEquals_BOOL(
	Expected 	:= inputStruct.expectedResult,
	Actual 		:= THIS^.assertorContainer.wasAssertionWrong,
	Message 	:= message
);
END_METHOD

(*

short summary
=============

.. <legal notes>

legal notes
=================
| SPDX-FileCopyrightText: © 2023 ekvip automation GmbH <info@ekvip.de>
| SPDX-License-Identifier: Apache-2.0
| For details check: Apache-2.0_

.. _Apache-2.0: https://www.apache.org/licenses/LICENSE-2.0

.. </legal notes>

parameters
==========

*)

{warning 'header is generated please add your documentation'}
METHOD testAsciiStartsWith : BOOL
VAR_INPUT
	inputStruct	: containsDataStr;
	testNumber 	: USINT;
END_VAR

VAR
	message : STRING;
END_VAR
THIS^.reset();

THIS^.assertorContainer.assertor.assert.strings.ascii.startsWith(
	stringToCheck	:= inputStruct.StringToTest,
	start			:= inputStruct.StringToContain,
	ignoreCases		:= inputStruct.IgnoreCases,
	trim			:= inputStruct.Trim,
	message			:= ''
);


message	:= CONCAT( 'Test Number ', TO_STRING(testNumber));
message	:= CONCAT( message, ' during function Ascii.startsWith ');
message	:= CONCAT( Message , ' has failed ');

THIS^.AssertEquals_BOOL(
	Expected 	:= inputStruct.expectedResult,
	Actual 		:= THIS^.assertorContainer.wasAssertionWrong,
	Message 	:= message
);
END_METHOD

(*

short summary
=============

.. <legal notes>

legal notes
=================
| SPDX-FileCopyrightText: © 2023 ekvip automation GmbH <info@ekvip.de>
| SPDX-License-Identifier: Apache-2.0
| For details check: Apache-2.0_

.. _Apache-2.0: https://www.apache.org/licenses/LICENSE-2.0

.. </legal notes>

parameters
==========

*)

{warning 'header is generated please add your documentation'}
METHOD testAsciiStringContains : BOOL
VAR_INPUT
	inputStruct	: containsDataStr;
	testNumber :USINT;
END_VAR

VAR
	message : STRING;
END_VAR
THIS^.reset();

THIS^.assertorContainer.assertor.assert.strings.ascii.contains(
	stringToCheck 	:= inputStruct.StringToTest,
	searchString	:= inputStruct.StringToContain, 
	ignoreCases		:= inputStruct.IgnoreCases,
	message         := ''
);

message	:= CONCAT( 'Test Number ', TO_STRING(testNumber));
message	:= CONCAT( message, ' during function Ascii.contains ');
message	:= CONCAT( Message , ' has failed ');

THIS^.AssertEquals_BOOL(
	Expected 	:= inputStruct.expectedResult,
	Actual 		:= THIS^.assertorContainer.wasAssertionWrong,
	Message 	:= message
);
END_METHOD

(*

short summary
=============

.. <legal notes>

legal notes
=================
| SPDX-FileCopyrightText: © 2023 ekvip automation GmbH <info@ekvip.de>
| SPDX-License-Identifier: Apache-2.0
| For details check: Apache-2.0_

.. _Apache-2.0: https://www.apache.org/licenses/LICENSE-2.0

.. </legal notes>

parameters
==========

*)

{warning 'header is generated please add your documentation'}
METHOD testAsciiStringContainsNo : BOOL
VAR_INPUT
	inputStruct	: containsDataStr;
	testNumber 	: USINT;
END_VAR

VAR
	message : STRING;
END_VAR
THIS^.reset();

THIS^.assertorContainer.assertor.assert.strings.utf16.containsNo(
	stringToCheck 	:= inputStruct.WStringToTest,
	searchString	:= inputStruct.WStringToContain, 
	ignoreCases		:= inputStruct.IgnoreCases,
	message         := ''
);

message	:= CONCAT( 'Test Number ', TO_STRING(testNumber));
message	:= CONCAT( message, ' during function Ascii.containsNo ');
message	:= CONCAT( Message , ' has failed ');

THIS^.AssertEquals_BOOL(
	Expected 	:= inputStruct.expectedResult,
	Actual 		:= THIS^.assertorContainer.wasAssertionWrong,
	Message 	:= message
);
END_METHOD

(*

short summary
=============

.. <legal notes>

legal notes
=================
| SPDX-FileCopyrightText: © 2023 ekvip automation GmbH <info@ekvip.de>
| SPDX-License-Identifier: Apache-2.0
| For details check: Apache-2.0_

.. _Apache-2.0: https://www.apache.org/licenses/LICENSE-2.0

.. </legal notes>

parameters
==========

*)

{warning 'header is generated please add your documentation'}
METHOD testAsciiStringLengthBetween
VAR_INPUT
	inputStruct	: IsLengthBetweenBasicData;
	testNumber 	: USINT;
END_VAR

VAR
	message : STRING;
END_VAR
THIS^.reset();

THIS^.assertorContainer.assertor.assert.strings.ascii.lenghtIsBetween( 
	stringToCheck	:=	inputStruct.stringToTest, 
	maxLenght		:=	inputStruct.maxLength,
	minLenght   	:=  inputStruct.minLength,
	message			:=	''          
);


message	:= CONCAT( 'Test Number ', TO_STRING(testNumber));
message	:= CONCAT( message, ' during function Ascii.isLengthBetween ');
message	:= CONCAT( Message , ' has failed ');
	
THIS^.AssertEquals_BOOL(
	Expected 	:= inputStruct.expectedResult,
	Actual 		:= THIS^.assertorContainer.wasAssertionWrong,
	Message 	:= message
);
END_METHOD

(*

short summary
=============

.. <legal notes>

legal notes
=================
| SPDX-FileCopyrightText: © 2023 ekvip automation GmbH <info@ekvip.de>
| SPDX-License-Identifier: Apache-2.0
| For details check: Apache-2.0_

.. _Apache-2.0: https://www.apache.org/licenses/LICENSE-2.0

.. </legal notes>

parameters
==========

*)

{warning 'header is generated please add your documentation'}
METHOD testAsciiStringlengthIs
VAR_INPUT
	inputStruct	:IsLengthBasicData;
	testNumber :USINT;
END_VAR

VAR
	message: STRING;
END_VAR

THIS^.reset();

IF (inputStruct.funcType = FunctionType.EXACT) THEN 
	THIS^.assertorContainer.assertor.assert.strings.ascii.lenghtIsExact( 
		stringToCheck	:=	inputStruct.stringToTest, 
		expectedLength	:=	TO_USINT(inputStruct.expectedLength),
		message			:=	''          
	);
ELSIF (inputStruct.funcType = FunctionType.MAXIMUM) THEN
	THIS^.assertorContainer.assertor.assert.strings.ascii.lenghtIsMax( 
		stringToCheck	:=	inputStruct.stringToTest, 
		maxLength		:=	TO_USINT(inputStruct.expectedLength),
		message			:=	''         
	);
ELSIF (inputStruct.funcType = FunctionType.MINIMUM) THEN
	THIS^.assertorContainer.assertor.assert.strings.ascii.lenghtIsMin( 
		stringToCheck	:=	inputStruct.stringToTest, 
		minLength		:=	TO_USINT(inputStruct.expectedLength),
		message			:=	''          
	);
END_IF;

message	:= CONCAT( 'Test Number ', TO_STRING(testNumber));
message	:= CONCAT( message, ' during function AsciiString.isLength ');
message	:= CONCAT( message , TO_STRING(inputStruct.funcType));
message	:= CONCAT( Message , ' has failed ');

THIS^.AssertEquals_BOOL(
	Expected 	:= inputStruct.expectedResult,
	Actual 		:= THIS^.assertorContainer.wasAssertionWrong,
	Message		:= message
);
END_METHOD

(*

short summary
=============

.. <legal notes>

legal notes
=================
| SPDX-FileCopyrightText: © 2023 ekvip automation GmbH <info@ekvip.de>
| SPDX-License-Identifier: Apache-2.0
| For details check: Apache-2.0_

.. _Apache-2.0: https://www.apache.org/licenses/LICENSE-2.0

.. </legal notes>

parameters
==========

*)

{warning 'header is generated please add your documentation'}
METHOD testUtf16EndsWith : BOOL
VAR_INPUT
	inputStruct	: containsDataStr;
	testNumber 	: USINT;
END_VAR

VAR
	message : STRING;
END_VAR
THIS^.reset();

THIS^.assertorContainer.assertor.assert.strings.utf16.endsWith(
	stringToCheck	:= inputStruct.WStringToTest,
	end				:= inputStruct.WStringToContain,
	ignoreCases		:= inputStruct.IgnoreCases,
	trim			:= inputStruct.Trim,
	message			:= ''
);

message	:= CONCAT( 'Test Number ', TO_STRING(testNumber));
message	:= CONCAT( message, ' during function UTF16.endsWith ');
message	:= CONCAT( Message , ' has failed ');

THIS^.AssertEquals_BOOL(
	Expected 	:= inputStruct.expectedResult,
	Actual 		:= THIS^.assertorContainer.wasAssertionWrong,
	Message 	:= message
);
END_METHOD

(*

short summary
=============

.. <legal notes>

legal notes
=================
| SPDX-FileCopyrightText: © 2023 ekvip automation GmbH <info@ekvip.de>
| SPDX-License-Identifier: Apache-2.0
| For details check: Apache-2.0_

.. _Apache-2.0: https://www.apache.org/licenses/LICENSE-2.0

.. </legal notes>

parameters
==========

*)

{warning 'header is generated please add your documentation'}
METHOD testUtf16IsEmpty : BOOL
VAR_INPUT
	inputStruct	: isEmptyDataStr;
	testNumber 	: USINT;
END_VAR

VAR
	message : STRING;
END_VAR
THIS^.reset();

THIS^.assertorContainer.assertor.assert.strings.anyString.isEmpty(
	stringToCheck 	:= inputStruct.WStringToTest,
	message			:= ''
);

message	:= CONCAT( 'Test Number ', TO_STRING(testNumber));
message	:= CONCAT( message, ' during function UTF16.isEmpty ');
message	:= CONCAT( Message , ' has failed ');

THIS^.AssertEquals_BOOL(
	Expected 	:= inputStruct.expectedResult,
	Actual 		:= THIS^.assertorContainer.wasAssertionWrong,
	Message 	:= message
);
END_METHOD

(*

short summary
=============

.. <legal notes>

legal notes
=================
| SPDX-FileCopyrightText: © 2023 ekvip automation GmbH <info@ekvip.de>
| SPDX-License-Identifier: Apache-2.0
| For details check: Apache-2.0_

.. _Apache-2.0: https://www.apache.org/licenses/LICENSE-2.0

.. </legal notes>

parameters
==========

*)

{warning 'header is generated please add your documentation'}
METHOD testUtf16IsEqualTo : BOOL
VAR_INPUT
	inputStruct	: isEqualToDataStr;
	testNumber 	: USINT;
END_VAR

VAR
	message : STRING;
END_VAR
THIS^.reset();

THIS^.assertorContainer.assertor.assert.strings.anyString.isEqualTo(
	stringToCheck 	:= inputStruct.WStringToTest,
	expected		:= inputStruct.EqualToWString,
	ignoreCases     := inputStruct.IgnoreCases,
	message			:= ''	 	
);
   
message	:= CONCAT( 'Test Number ', TO_STRING(testNumber));
message	:= CONCAT( message, ' during function UTF16.isEqualTo ');
message	:= CONCAT( Message , ' has failed ');

THIS^.AssertEquals_BOOL(
	Expected 	:= inputStruct.expectedResult,
	Actual 		:= THIS^.assertorContainer.wasAssertionWrong,
	Message 	:= message
);
END_METHOD

(*

short summary
=============

.. <legal notes>

legal notes
=================
| SPDX-FileCopyrightText: © 2023 ekvip automation GmbH <info@ekvip.de>
| SPDX-License-Identifier: Apache-2.0
| For details check: Apache-2.0_

.. _Apache-2.0: https://www.apache.org/licenses/LICENSE-2.0

.. </legal notes>

parameters
==========

*)

{warning 'header is generated please add your documentation'}
METHOD testUtf16IsNotEmpty : BOOL
VAR_INPUT
	inputStruct	: isEmptyDataStr;
	testNumber 	: USINT;
END_VAR

VAR
	message : STRING;
END_VAR
THIS^.reset();

THIS^.assertorContainer.assertor.assert.strings.anyString.isNotEmpty(
	stringToCheck 	:= inputStruct.WStringToTest,
	message			:= ''
);

message	:= CONCAT( 'Test Number ', TO_STRING(testNumber));
message	:= CONCAT( message, ' during function UTF16.isNotEmpty ');
message	:= CONCAT( Message , ' has failed ');

THIS^.AssertEquals_BOOL(
	Expected 	:= inputStruct.expectedResult,
	Actual 		:= THIS^.assertorContainer.wasAssertionWrong,
	Message 	:= message
);
END_METHOD

(*

short summary
=============

.. <legal notes>

legal notes
=================
| SPDX-FileCopyrightText: © 2023 ekvip automation GmbH <info@ekvip.de>
| SPDX-License-Identifier: Apache-2.0
| For details check: Apache-2.0_

.. _Apache-2.0: https://www.apache.org/licenses/LICENSE-2.0

.. </legal notes>

parameters
==========

*)

{warning 'header is generated please add your documentation'}
METHOD testUtf16IsNotEqualTo : BOOL
VAR_INPUT
	inputStruct	: isEqualToDataStr;
	testNumber 	: USINT;
END_VAR

VAR
	message : STRING;
END_VAR
THIS^.reset();

THIS^.assertorContainer.assertor.assert.strings.anyString.isNotEqualTo(
	stringToCheck 	:= inputStruct.WStringToTest,
	unexpected		:= inputStruct.EqualToWString,
	ignoreCases     := inputStruct.IgnoreCases,
	message			:= ''	 	
);
   
message	:= CONCAT( 'Test Number ', TO_STRING(testNumber));
message	:= CONCAT( message, ' during function UTF16.isNotEqualTo ');
message	:= CONCAT( Message , ' has failed ');

THIS^.AssertEquals_BOOL(
	Expected 	:= inputStruct.expectedResult,
	Actual 		:= THIS^.assertorContainer.wasAssertionWrong,
	Message 	:= message
);
END_METHOD

(*

short summary
=============

.. <legal notes>

legal notes
=================
| SPDX-FileCopyrightText: © 2023 ekvip automation GmbH <info@ekvip.de>
| SPDX-License-Identifier: Apache-2.0
| For details check: Apache-2.0_

.. _Apache-2.0: https://www.apache.org/licenses/LICENSE-2.0

.. </legal notes>

parameters
==========

*)

{warning 'header is generated please add your documentation'}
METHOD testUtf16StartsWith : BOOL
VAR_INPUT
	inputStruct	: containsDataStr;
	testNumber 	: USINT;
END_VAR

VAR
	message : STRING;
END_VAR
THIS^.reset();

THIS^.assertorContainer.assertor.assert.strings.utf16.startsWith(
	stringToCheck	:= inputStruct.WStringToTest,
	start			:= inputStruct.WStringToContain,
	ignoreCases		:= inputStruct.IgnoreCases,
	trim			:= inputStruct.Trim,
	message			:= ''
);

message	:= CONCAT( 'Test Number ', TO_STRING(testNumber));
message	:= CONCAT( message, ' during function UTF16.startsWith ');
message	:= CONCAT( Message , ' has failed ');

THIS^.AssertEquals_BOOL(
	Expected 	:= inputStruct.expectedResult,
	Actual 		:= THIS^.assertorContainer.wasAssertionWrong,
	Message 	:= message
);
END_METHOD

(*

short summary
=============

.. <legal notes>

legal notes
=================
| SPDX-FileCopyrightText: © 2023 ekvip automation GmbH <info@ekvip.de>
| SPDX-License-Identifier: Apache-2.0
| For details check: Apache-2.0_

.. _Apache-2.0: https://www.apache.org/licenses/LICENSE-2.0

.. </legal notes>

parameters
==========

*)

{warning 'header is generated please add your documentation'}
METHOD testUtf16StringContains : BOOL
VAR_INPUT
	inputStruct	: containsDataStr;
	testNumber :USINT;
END_VAR

VAR
	message : STRING;
END_VAR
THIS^.reset();

THIS^.assertorContainer.assertor.assert.strings.utf16.contains(
	stringToCheck 	:= inputStruct.WStringToTest,
	searchString	:= inputStruct.WStringToContain, 
	ignoreCases		:= inputStruct.IgnoreCases,
	message         := ''
);

message	:= CONCAT( 'Test Number ', TO_STRING(testNumber));
message	:= CONCAT( message, ' during function UTF16.contains ');
message	:= CONCAT( Message , ' has failed ');

THIS^.AssertEquals_BOOL(
	Expected 	:= inputStruct.expectedResult,
	Actual 		:= THIS^.assertorContainer.wasAssertionWrong,
	Message 	:= message
);
END_METHOD

(*

short summary
=============

.. <legal notes>

legal notes
=================
| SPDX-FileCopyrightText: © 2023 ekvip automation GmbH <info@ekvip.de>
| SPDX-License-Identifier: Apache-2.0
| For details check: Apache-2.0_

.. _Apache-2.0: https://www.apache.org/licenses/LICENSE-2.0

.. </legal notes>

parameters
==========

*)

{warning 'header is generated please add your documentation'}
METHOD testUtf16StringContainsNo : BOOL
VAR_INPUT
	inputStruct	: containsDataStr;
	testNumber 	: USINT;
END_VAR

VAR
	message : STRING;
END_VAR
THIS^.reset();

THIS^.assertorContainer.assertor.assert.strings.utf16.containsNo(
	stringToCheck 	:= inputStruct.WStringToTest,
	searchString	:= inputStruct.WStringToContain, 
	ignoreCases		:= inputStruct.IgnoreCases,
	message         := ''
);

message	:= CONCAT( 'Test Number ', TO_STRING(testNumber));
message	:= CONCAT( message, ' during function UTF16.containsNo ');
message	:= CONCAT( Message , ' has failed ');

THIS^.AssertEquals_BOOL(
	Expected 	:= inputStruct.expectedResult,
	Actual 		:= THIS^.assertorContainer.wasAssertionWrong,
	Message 	:= message
);
END_METHOD

(*

short summary
=============

.. <legal notes>

legal notes
=================
| SPDX-FileCopyrightText: © 2023 ekvip automation GmbH <info@ekvip.de>
| SPDX-License-Identifier: Apache-2.0
| For details check: Apache-2.0_

.. _Apache-2.0: https://www.apache.org/licenses/LICENSE-2.0

.. </legal notes>

parameters
==========

*)

{warning 'header is generated please add your documentation'}
METHOD testUtf16StringLengthBetween
VAR_INPUT
	inputStruct : IsLengthBetweenBasicData;
	testNumber	: USINT;
END_VAR

VAR
	message: STRING;
END_VAR
THIS^.reset();

THIS^.assertorContainer.assertor.assert.strings.utf16.lenghtIsBetween( 
	stringToCheck	:=	inputStruct.wstringToTest, 
	maxLenght		:=	inputStruct.maxLength,
	minLenght   	:=  inputStruct.minLength,
	message			:=	''          
);


message	:= CONCAT( 'Test Number ', TO_STRING(testNumber));
message	:= CONCAT( message, ' during function UTF16.isLengthBetween ');
message	:= CONCAT( Message , ' has failed ');
	
THIS^.AssertEquals_BOOL(
	Expected 	:= inputStruct.expectedResult,
	Actual 		:= THIS^.assertorContainer.wasAssertionWrong,
	Message 	:= message
);
END_METHOD

(*

short summary
=============

.. <legal notes>

legal notes
=================
| SPDX-FileCopyrightText: © 2023 ekvip automation GmbH <info@ekvip.de>
| SPDX-License-Identifier: Apache-2.0
| For details check: Apache-2.0_

.. _Apache-2.0: https://www.apache.org/licenses/LICENSE-2.0

.. </legal notes>

parameters
==========

*)

{warning 'header is generated please add your documentation'}
METHOD testUtf16StringlengthIs
VAR_INPUT
	inputStruct	:IsLengthBasicData;
	testNumber :USINT;
END_VAR

VAR
	message: STRING;
END_VAR

THIS^.reset();

IF (inputStruct.funcType = FunctionType.EXACT) THEN
	THIS^.assertorContainer.assertor.assert.strings.utf16.lenghtIsExact( 
		stringToCheck	:=	inputStruct.wstringToTest, 
		expectedLength	:=	TO_USINT(inputStruct.expectedLength),
		message			:=	''          
	);
ELSIF (inputStruct.funcType = FunctionType.MAXIMUM) THEN
	THIS^.assertorContainer.assertor.assert.strings.utf16.lenghtIsMax( 
		stringToCheck	:=	inputStruct.wstringToTest, 
		maxLength		:=	TO_USINT(inputStruct.expectedLength),
		message			:=	''         
	);
ELSIF (inputStruct.funcType = FunctionType.MINIMUM) THEN
	THIS^.assertorContainer.assertor.assert.strings.utf16.lenghtIsMin( 
		stringToCheck	:=	inputStruct.wstringToTest, 
		minLength		:=	TO_USINT(inputStruct.expectedLength),
		message			:=	' '         
	);
END_IF;

message	:= CONCAT( ' Test Number ', TO_STRING(testNumber));
message	:= CONCAT( message, ' during function UFT16String.isLength ');
message	:= CONCAT( message , TO_STRING(inputStruct.funcType));
message	:= CONCAT( Message , ' has failed ');
	
THIS^.AssertEquals_BOOL(
	Expected 	:= inputStruct.expectedResult,
	Actual 		:= THIS^.assertorContainer.wasAssertionWrong,
	Message 	:= message
);
END_METHOD

END_FUNCTION_BLOCK

(* stored: Version 1.1.0.1, ProductVersion 3.1.4024.12
   POU StringAssertionTests: Id {ef77a513-4fcf-4f2c-86b9-4cd7add41495}, SpecialFunc None
   Folder anyString: Id {326b4f68-416f-4510-aae7-68b0da96aefb}
   Folder contains: Id {9474e84a-b84d-4c31-b0a2-e15604db1a06}
   Folder containsNo: Id {420e7f08-5049-44a4-9734-edfcca81f37c}
   Folder endsWith: Id {b00bee8f-398a-4b88-a437-ace63a5fe11c}
   Folder isEmpty: Id {bc905500-581b-4370-be28-5abca9180009}
   Folder isEqualTo: Id {5a70313a-d317-4b5a-99c9-87a59f45056c}
   Folder isLenghtExact: Id {72195a71-537a-4e07-96e1-9e07c5705a02}
   Folder isLengthBetween: Id {1e7cabdc-b378-4466-a2a0-23775041abd6}
   Folder isNotEmpty: Id {0edcf8c0-85c3-4b23-8872-a498606f3996}
   Folder isNotEqualTo: Id {6f396fc0-265b-4f83-bdf0-687beb929d7a}
   Folder startsWith: Id {0aba82d7-f1d6-4728-9aa8-223e7d9a1c89}
   Method FB_init: Id {37f790e4-9b93-41b6-874e-7819cf1e1351}
   Method reset: Id {c76d3913-e022-4ce3-a266-16e157e59c0b}
   Method runTestContains: Id {8f886456-c87a-4b48-801a-7b98beae770c}
   Method runTestContainsNo: Id {032e8792-a8e8-48df-9e1b-7b1a8e065719}
   Method runTestEndsWith: Id {8473644e-5a41-43a2-b1d3-4da733f8832b}
   Method runTestIsEmpty: Id {0199bc09-5ad2-4022-b544-b00ae894a785}
   Method runTestIsEqualTo: Id {1a17c691-080f-4193-8c9f-3b6be8f3e80d}
   Method runTestIsLength: Id {f13bc3b9-26f3-43d4-a4cd-b43a2c2ff682}
   Method runTestIsNotEmpty: Id {03d1da4c-b365-44a6-875c-c1cea05ba4ee}
   Method runTestIsNotEqualTo: Id {f589512f-d22c-41b2-915f-a8f19ec9a9fe}
   Method runTestLengthIsBetween: Id {1e1519eb-6e8e-47e7-8611-90a898f0a977}
   Method runTestStartsWith: Id {7bc18a33-2123-4d4d-b680-2b949689b55f}
   Method testAnyString_isEmpty: Id {9a09f0a9-8be8-4f02-a68a-5b0d4467e103}
   Method testAnyString_isEqualTo: Id {5a48ae37-fa18-47cf-928d-3d7690b9d09e}
   Method testAnyString_isNotEmpty: Id {c5a98256-6ef3-48ea-97c0-ec0b37b2e81c}
   Method testAnyString_isNotEqualTo: Id {6601a9bd-02d3-4d43-973e-4c7500ab7c9d}
   Method testAnyString_lengthIsExact: Id {4bb7aa35-39f2-483b-b247-5c9edfe867af}
   Method testAnyStringContains: Id {74e905da-faff-4755-b6cc-57fbc37b8493}
   Method testAnyStringContainsNo: Id {a578bd77-1b34-437f-9ddb-49b804b292dc}
   Method testAnyStringEndsWith: Id {db544b7a-b433-4aa9-a93c-3044c971dd76}
   Method testAnyStringIsEmpty: Id {ceab1f12-94cd-49ba-a4cf-66ddce7eabaa}
   Method testAnyStringIsEqualTo: Id {fe41d322-4945-4d44-8259-ffa5ce44d1ac}
   Method testAnyStringIsNotEmpty: Id {bdc4e7b2-8b10-48bb-96f7-b24468ce9b1f}
   Method testAnyStringIsNotEqualTo: Id {1e544c79-a5de-484b-8e67-bc76c5272806}
   Method testAnyStringLengthBetween: Id {420a62d6-64f2-48ea-9dc6-3bec23023bdf}
   Method testAnyStringLengthIs: Id {eb8f4deb-44b3-487b-937f-1e3b2e61a4c4}
   Method testAnyStringStartsWith: Id {2165e8b2-f15d-41ac-aa27-87c2f35b62f4}
   Method testAsciiEndsWith: Id {6309f128-8053-43ef-a8cb-fbcd7d1539d5}
   Method testAsciiIsEmpty: Id {1e895922-1fbc-481a-abe2-f69bb2c677f0}
   Method testAsciiIsEqualTo: Id {1c7f9bb9-4da8-47f4-be1b-5dfddf7d7d74}
   Method testAsciiIsNotEmpty: Id {f57de34a-f4df-446a-803c-77b9579706cf}
   Method testAsciiIsNotEqualTo: Id {a0c73e4c-3bde-468c-a486-3deaa98cd4d5}
   Method testAsciiStartsWith: Id {c51554cf-d9cc-4f5a-b0ea-acfc8629f5d1}
   Method testAsciiStringContains: Id {5403121a-a2f1-424f-ae7f-32e7f0066deb}
   Method testAsciiStringContainsNo: Id {b8bade71-f498-47ed-9d19-a1ac5ad28643}
   Method testAsciiStringLengthBetween: Id {ddbebe76-9b96-4b67-bd40-db8b5f2518a1}
   Method testAsciiStringlengthIs: Id {33c8ffbf-97d8-4e59-a10a-936b759ed63c}
   Method testUtf16EndsWith: Id {e890ec3d-cd18-4716-8a10-a10c86b1920f}
   Method testUtf16IsEmpty: Id {b61ab6be-2063-4be7-823a-d82d64c09b38}
   Method testUtf16IsEqualTo: Id {0ccc7132-2a60-4465-875e-5484a68209cf}
   Method testUtf16IsNotEmpty: Id {8f253903-a43a-4961-81a1-0ec659194759}
   Method testUtf16IsNotEqualTo: Id {87540caf-b339-4568-886e-66d16808b29f}
   Method testUtf16StartsWith: Id {9324069b-dd77-44fd-8a32-89ad628489c5}
   Method testUtf16StringContains: Id {b44ec857-bbed-48b4-92c6-7868702c1646}
   Method testUtf16StringContainsNo: Id {e82994f3-0f6d-40a0-b47c-5d7f344d79f4}
   Method testUtf16StringLengthBetween: Id {715641ec-876e-471f-b535-347afb0424b7}
   Method testUtf16StringlengthIs: Id {040791d6-e31e-4fae-a77f-1b1be34964e8} *)
